(* IEC 61131-3 sources: std_i2980_v2.06_cp053/Source/IMM/ieccontrol/system (part 2) *)

(* ---- ABEnergy.pu ---- *)
(*
@h    ! WARNING !
@h    The Kemro K2 system (including software) only meets category B according to EN 954-1,
@h    thus it is not intended for usage in safety-relevant control applications in the field
@h    of personal safety (e.g. emergency stop).
@h    To implement potentially necessary safety-relevant control tasks, always use additional
@h    external safety devices that are intended for the particular purpose, and meet the necessary
@h    functional safety.
@h    For further information see EN 954-1 (EN ISO 13849-1) and/or the K2-x00 user manual, chapter
@h    "CE conformity, directives and standards".

This AB calculate the energy.

*)

IMPORT_OVER_LISTFILE
 GET_SYNC_REFTO
, GET_TASK_INTERVAL
, GET_MY_FU_NAME
, KSWO_AddVariable
, START_PROCESS_ALGORITHM
, STOP_PROCESS_ALGORITHM
, KSYS_Status_OK
, nHalfAutomatic
, nFullAutomatic
, cCompEnergyMeter
, tnOperationMode
, tyNumberOfDevices
, KSYS_Status
, KSWO_Status

END_IMPORT

ALGORITHM_BLOCK ABEnergy #DUMMY_EDIT_BLOCK

SYSTEM_VAR
 sv_bResetShotCounter : BOOL (* reset shot counter *);
 sv_iProdCounterAct : DINT;
 sv_iShotCounterAct : DINT;
 sv_rEnergyShot : REAL (* energy per shot *);
 sv_rEnergyProduction : REAL (* energy per production *);
 sv_rEnergyPart : REAL (* energy per part *);
 sv_rEnergyShotVolume : REAL (* energy in shot volume *);
 sv_rEnergyPartMass : REAL (* energy in part mass *);
 sv_rPartMass : REAL (* part mass *);
 sv_rHeatingPower : REAL (* heating power *);
 sv_rTotalEnergy : REAL (* total energy *);
 sv_rTotalPower : REAL (* total power *);
 sv_rMotorPower : REAL (* motor power *);
 sv_bResetTotEnergy : BOOL (* reset energy *);
 sv_OperationMode : tnOperationMode;
 sv_bStartSampleMeasure : BOOL;
 sv_rSampleMeasuredEnergy : REAL;
 sv_iAutoStopShotCounter : DINT;
 sv_dMeasuredDuration : TIME (* measured duration in mins  *);
 sv_dSetDuration : TIME (* set duration for sample energy measurement in mins  *);
 sv_rMeasuredPower : REAL (* measured  power *);
 sv_rMeasuredEnergy : REAL (* measured energy *);
 sv_rTotalEnergyCalibrated : REAL (* total energy *);
 sv_rTotalPowerCalibrated : REAL (* total power *);
 sv_rIdlePower : REAL;
 sv_rMeasuredEnergyHMI : REAL;
 sv_NumberOfDevices : tyNumberOfDevices;
 sv_bInitDone : BOOL;
 sv_rEfficiency : REAL;
END_VAR

SYSTEM_OBJECT
 TaskMid : TASK;
 TaskSlow : TASK;
 TaskHeating : TASK;
 TaskInject : TASK;
 PU_Task_7 : TASK;
END_OBJECT

VAR
 mrMotorPower : REAL;
 mprActCushion : REFTO REAL;
 mprCushionZeroPosition : REFTO REAL;
 mrActEnergy : REAL;
 mrTotEnergyLastShot : REAL;
 mrTotEnergyLastPart : REAL;
 mrShotVolume : REAL;
 mrTmpEnergy : REAL;
 mrLastActEnergy : REAL;
 mprHeatingPowerNozzle1 : REFTO REAL;
 mprHeatingPowerMold1 : REFTO REAL;
 mbHeatingPowerNozzle1Linked : BOOL;
 mbHeatingPowerMold1Linked : BOOL;
 mrRecordedEnergy : REAL;
 mbCycleRestarted : BOOL;
 miShotCounter : DINT;
 mrRecordedSampleEnergy : REAL;
 mrActEnergyCalibrated : REAL;
 mrTmpEnergyCalibrated : REAL;
 mbEnergyMeterLinked : BOOL;
 mprMotorPowerSpeedpump : REFTO REAL;
 mprMotorPowerEject : REFTO REAL;
 mprMotorPowerInject : REFTO REAL;
 mprMotorPowerPlast : REFTO REAL;
 mprMotorPowerMold : REFTO REAL;
 mprMotorPowerNozzle : REFTO REAL;
END_VAR

(*
@h    ! WARNING !
@h    The Kemro K2 system (including software) only meets category B according to EN 954-1,
@h    thus it is not intended for usage in safety-relevant control applications in the field
@h    of personal safety (e.g. emergency stop).
@h    To implement potentially necessary safety-relevant control tasks, always use additional
@h    external safety devices that are intended for the particular purpose, and meet the necessary
@h    functional safety.
@h    For further information see EN 954-1 (EN ISO 13849-1) and/or the K2-x00 user manual, chapter
@h    "CE conformity, directives and standards".

This algo initializes for the energy calculation

*)

PROCESS_ALGORITHM paInit ON TaskMid AUTOSTART

VAR
 Status : KSYS_Status;
END_VAR
#BEGIN_EDIT_BLOCK
(**************************************** WARNING ********************************************
 *** The KEBA Kemro K2 System including software is not intended for safety control tasks! ***
 ***                       For further information see Comment tab!                        ***
 *********************************************************************************************)

(*pointer to motor total power speedpump*)
mprMotorPowerSpeedpump := GET_SYNC_REFTO('Pump1.sv_rMotorTotalPower', T#0s, Status);

IF Status <> KSYS_Status_OK  THEN
   mprMotorPowerSpeedpump := GET_SYNC_REFTO('system.sv_rNull', T#0s, Status);
END_IF;

(*pointer to motor power elec.axes*)
mprMotorPowerEject := GET_SYNC_REFTO('Ejector1.sv_rMotorPowerEject', T#0s, Status);
IF Status <> KSYS_Status_OK  THEN
   mprMotorPowerEject := GET_SYNC_REFTO('system.sv_rNull', T#0s, Status);
END_IF;

mprMotorPowerInject:= GET_SYNC_REFTO('Injection1.sv_rMotorPowerInject', T#0s, Status);
IF Status <> KSYS_Status_OK  THEN
   mprMotorPowerInject := GET_SYNC_REFTO('system.sv_rNull', T#0s, Status);
END_IF;

mprMotorPowerPlast:= GET_SYNC_REFTO('Injection1.sv_rMotorPowerPlast', T#0s, Status);
IF Status <> KSYS_Status_OK  THEN
   mprMotorPowerPlast := GET_SYNC_REFTO('system.sv_rNull', T#0s, Status);
END_IF;

mprMotorPowerMold:= GET_SYNC_REFTO('Mold1.sv_rMotorPowerMold', T#0s, Status);
IF Status <> KSYS_Status_OK  THEN
   mprMotorPowerMold := GET_SYNC_REFTO('system.sv_rNull', T#0s, Status);
END_IF;

mprMotorPowerNozzle:= GET_SYNC_REFTO('Nozzle1.sv_rMotorPowerNozzle', T#0s, Status);
IF Status <> KSYS_Status_OK  THEN
   mprMotorPowerNozzle := GET_SYNC_REFTO('system.sv_rNull', T#0s, Status);
END_IF;

mprActCushion := GET_SYNC_REFTO('Injection1.sv_rCushion', T#0s, Status);
mprCushionZeroPosition := GET_SYNC_REFTO('Injection1.sv_rScrewZeroPosition', T#0s, Status);

mprHeatingPowerNozzle1 := GET_SYNC_REFTO('HeatingNozzle1.sv_rActHeatingPower', T#0s, Status);
IF Status = KSYS_Status_OK THEN
   mbHeatingPowerNozzle1Linked := TRUE;
END_IF;
mprHeatingPowerMold1 := GET_SYNC_REFTO('HeatingMold1.sv_rActHeatingPower', T#0s, Status);
IF Status = KSYS_Status_OK THEN
   mbHeatingPowerMold1Linked := TRUE;
END_IF;

STOP_PROCESS_ALGORITHM();

;#END_EDIT_BLOCK END_ALGORITHM

(*
@h    ! WARNING !
@h    The Kemro K2 system (including software) only meets category B according to EN 954-1,
@h    thus it is not intended for usage in safety-relevant control applications in the field
@h    of personal safety (e.g. emergency stop).
@h    To implement potentially necessary safety-relevant control tasks, always use additional
@h    external safety devices that are intended for the particular purpose, and meet the necessary
@h    functional safety.
@h    For further information see EN 954-1 (EN ISO 13849-1) and/or the K2-x00 user manual, chapter
@h    "CE conformity, directives and standards".

This postupdate algorithms calculates the energy per shot and per ccm.

*)

POSTUPDATE_ALGORITHM pCalcEnergyShot ON TaskMid WITH sv_iShotCounterAct

#BEGIN_EDIT_BLOCK
(**************************************** WARNING ********************************************
 *** The KEBA Kemro K2 System including software is not intended for safety control tasks! ***
 ***                       For further information see Comment tab!                        ***
 *********************************************************************************************)

(*Calculation of the energy cosumption per shot*)
sv_rEnergyShot := mrActEnergy - mrTotEnergyLastShot;
mrTotEnergyLastShot := mrActEnergy;

(*Calculation of the energy cosumption per ccm*)
mrShotVolume := mprCushionZeroPosition^ - mprActCushion^;  (*calculate the shot volume*)

IF mrShotVolume <> 0.0 THEN
  sv_rEnergyShotVolume := sv_rEnergyShot / mrShotVolume;
ELSE
  sv_rEnergyShotVolume := 0.0;
END_IF;

//Synchronization to machine cycle
IF mbEnergyMeterLinked THEN
  IF sv_bStartSampleMeasure THEN

  //start the sample measurement
    IF NOT mbCycleRestarted THEN
      mbCycleRestarted := TRUE;
    END_IF;

    //shot counter for the sample measurement
    miShotCounter := miShotCounter + 1;
    END_IF;
END_IF;

;#END_EDIT_BLOCK END_ALGORITHM

(*
@h    ! WARNING !
@h    The Kemro K2 system (including software) only meets category B according to EN 954-1,
@h    thus it is not intended for usage in safety-relevant control applications in the field
@h    of personal safety (e.g. emergency stop).
@h    To implement potentially necessary safety-relevant control tasks, always use additional
@h    external safety devices that are intended for the particular purpose, and meet the necessary
@h    functional safety.
@h    For further information see EN 954-1 (EN ISO 13849-1) and/or the K2-x00 user manual, chapter
@h    "CE conformity, directives and standards".

This AB calculates the energy per production.

*)

POSTUPDATE_ALGORITHM pUpdateEnergyProduction ON TaskMid WITH sv_bResetShotCounter

#BEGIN_EDIT_BLOCK
(**************************************** WARNING ********************************************
 *** The KEBA Kemro K2 System including software is not intended for safety control tasks! ***
 ***                       For further information see Comment tab!                        ***
 *********************************************************************************************)
sv_rEnergyProduction := 0.0;             (*reset the energy per production*)
mrLastActEnergy := mrActEnergy;          (*copy the calculated energy of the last cycle*)

;#END_EDIT_BLOCK END_ALGORITHM

(*
@h    ! WARNING !
@h    The Kemro K2 system (including software) only meets category B according to EN 954-1,
@h    thus it is not intended for usage in safety-relevant control applications in the field
@h    of personal safety (e.g. emergency stop).
@h    To implement potentially necessary safety-relevant control tasks, always use additional
@h    external safety devices that are intended for the particular purpose, and meet the necessary
@h    functional safety.
@h    For further information see EN 954-1 (EN ISO 13849-1) and/or the K2-x00 user manual, chapter
@h    "CE conformity, directives and standards".

This postupdate algorithm calculates the energy per gram.
*)

POSTUPDATE_ALGORITHM pCalcEnergyPart ON TaskMid WITH sv_iProdCounterAct,sv_rPartMass

#BEGIN_EDIT_BLOCK
(**************************************** WARNING ********************************************
 *** The KEBA Kemro K2 System including software is not intended for safety control tasks! ***
 ***                       For further information see Comment tab!                        ***
 *********************************************************************************************)

(*Calculation of the energy cosumption per part*)
sv_rEnergyPart := mrActEnergy - mrTotEnergyLastPart;
mrTotEnergyLastPart := mrActEnergy;

(*Calculation of the energy cosumption in part mass*)
IF sv_rPartMass <> 0.0 THEN
    sv_rEnergyPartMass := sv_rEnergyPart / sv_rPartMass;
ELSE
    sv_rEnergyPartMass := 0.0;
END_IF;

;#END_EDIT_BLOCK END_ALGORITHM

(*
@h    ! WARNING !
@h    The Kemro K2 system (including software) only meets category B according to EN 954-1,
@h    thus it is not intended for usage in safety-relevant control applications in the field
@h    of personal safety (e.g. emergency stop).
@h    To implement potentially necessary safety-relevant control tasks, always use additional
@h    external safety devices that are intended for the particular purpose, and meet the necessary
@h    functional safety.
@h    For further information see EN 954-1 (EN ISO 13849-1) and/or the K2-x00 user manual, chapter
@h    "CE conformity, directives and standards".

This process algorithm calculates the energy.
*)

PROCESS_ALGORITHM paCalcAndMeasure ON TaskHeating

VAR_TEMP
 b : BOOL;
END_VAR

VAR
 rHeatingPower : REAL;
 dCycleTime : TIME;
 bInitDone : BOOL;
 rCycleTime : REAL;
END_VAR
#BEGIN_EDIT_BLOCK
(**************************************** WARNING ********************************************
 *** The KEBA Kemro K2 System including software is not intended for safety control tasks! ***
 ***                       For further information see Comment tab!                        ***
 *********************************************************************************************)

(* Cycle time *)
IF NOT bInitDone THEN
   dCycleTime := GET_TASK_INTERVAL();
   rCycleTime := (LINT_TO_REAL(TIME_TO_LINT(dCycleTime))) / 1000000.0;
   bInitDone := TRUE;
END_IF;

(* Motor power estimated [kW] *)
mrMotorPower :=  mprMotorPowerSpeedpump^ +  mprMotorPowerEject^ +  mprMotorPowerInject^ +  mprMotorPowerPlast^ + mprMotorPowerMold^ + mprMotorPowerNozzle^;
b := WRITE_SVREAL_DIRECT(sv_rMotorPower, mrMotorPower);

(* Heat power estimated [W] *)
rHeatingPower := 0.0;
IF mbHeatingPowerNozzle1Linked THEN
   rHeatingPower := rHeatingPower + mprHeatingPowerNozzle1^;
END_IF;
IF mbHeatingPowerMold1Linked THEN
   rHeatingPower := rHeatingPower + mprHeatingPowerMold1^;
END_IF;
b := WRITE_SVREAL_DIRECT(sv_rHeatingPower, rHeatingPower);

(* Total power [kW] *)
IF mbEnergyMeterLinked THEN
   //Calculate the total power from measured total power
   b := WRITE_SVREAL_DIRECT(sv_rTotalPower, (sv_rMeasuredPower / 1000.0));
ELSE
   b := WRITE_SVREAL_DIRECT(sv_rTotalPower, (((rHeatingPower + sv_rIdlePower) / 1000.0 + mrMotorPower) / sv_rEfficiency));
END_IF;

(* Energy *)
IF mbEnergyMeterLinked THEN
   (* Total energy from power meter [kwh] *)
   sv_rTotalEnergy := (sv_rMeasuredEnergy - mrRecordedEnergy) / 1000.0; //measured value in Wh
   mrActEnergy := sv_rTotalEnergy;
   b := WRITE_SVREAL_DIRECT(sv_rMeasuredEnergyHMI, (sv_rMeasuredEnergy / 1000.0));

   (* Calculate the energy per production [kwh] *)
   IF sv_OperationMode >= nHalfAutomatic THEN
      b := WRITE_SVREAL_DIRECT(sv_rEnergyProduction, ((mrActEnergy - mrLastActEnergy) / 1000.0));
   END_IF;
ELSE
   (* Integration of power = Energy [kWs] *)
   mrActEnergy := mrTmpEnergy + sv_rTotalPower * rCycleTime;
   mrTmpEnergy := mrActEnergy;

   (* Calculate the energy per production [kwh] *)
   IF sv_OperationMode >= nHalfAutomatic THEN
      b := WRITE_SVREAL_DIRECT(sv_rEnergyProduction, ((mrActEnergy - mrLastActEnergy) / 3600.0));
   END_IF;

   (* Consumption of energy [kwh] *)
   sv_rTotalEnergy := (mrActEnergy / 3600.0 + mrRecordedEnergy);
END_IF;

(* Calibration *)
IF mbEnergyMeterLinked THEN
   (* Power calibration *)
   b := WRITE_SVREAL_DIRECT(sv_rTotalPowerCalibrated, ((sv_rMotorPower + (sv_rHeatingPower + sv_rIdlePower) / 1000.0) / sv_rEfficiency));

   (* Energy calibration *)
   mrActEnergyCalibrated := mrTmpEnergyCalibrated + sv_rTotalPowerCalibrated * rCycleTime;
   mrTmpEnergyCalibrated := mrActEnergyCalibrated;
   b := WRITE_SVREAL_DIRECT(sv_rTotalEnergyCalibrated, (mrActEnergyCalibrated / 3600.0));
END_IF;

;#END_EDIT_BLOCK END_ALGORITHM

(*
@h    ! WARNING !
@h    The Kemro K2 system (including software) only meets category B according to EN 954-1,
@h    thus it is not intended for usage in safety-relevant control applications in the field
@h    of personal safety (e.g. emergency stop).
@h    To implement potentially necessary safety-relevant control tasks, always use additional
@h    external safety devices that are intended for the particular purpose, and meet the necessary
@h    functional safety.
@h    For further information see EN 954-1 (EN ISO 13849-1) and/or the K2-x00 user manual, chapter
@h    "CE conformity, directives and standards".

This postupdate algorithm resets the energy calculation.
*)

POSTUPDATE_ALGORITHM pResetTotalEnergy ON TaskMid WITH sv_bResetTotEnergy

#BEGIN_EDIT_BLOCK
(**************************************** WARNING ********************************************
 *** The KEBA Kemro K2 System including software is not intended for safety control tasks! ***
 ***                       For further information see Comment tab!                        ***
 *********************************************************************************************)
(*reset the energy calculator*)
IF sv_bResetTotEnergy THEN
   //when power meter is used, record the last measured total energy,
   //and calculate always the difference between the actual measured value and recorded value
   //when estimation is used, integration of power with initial value 0 would be restarted
   IF mbEnergyMeterLinked THEN
     mrRecordedEnergy := sv_rMeasuredEnergy;
   ELSE
     mrRecordedEnergy := 0.0;
   END_IF;

   mrActEnergy := 0.0;
   mrTmpEnergy := 0.0;
   sv_rTotalEnergy := 0.0;
   mrLastActEnergy := 0.0;
   mrTotEnergyLastShot := 0.0;
   mrTotEnergyLastPart := 0.0;
   sv_bResetTotEnergy := FALSE;

   //calibration
   IF mbEnergyMeterLinked THEN
     mrActEnergyCalibrated := 0.0;
     mrTmpEnergyCalibrated := 0.0;
     sv_rTotalEnergyCalibrated := 0.0;
   END_IF;
END_IF;

;#END_EDIT_BLOCK END_ALGORITHM

PROCESS_ALGORITHM paInitDebugMeasurement ON TaskSlow AUTOSTART

VAR
 fuName : STRING(255);
 variableName : STRING(255);
 swoState : KSWO_Status;
END_VAR
#BEGIN_EDIT_BLOCK
(**************************************** WARNING ********************************************
 *** The KEBA Kemro K2 System including software is not intended for safety control tasks! ***
 ***                       For further information see Comment tab!                        ***
 *********************************************************************************************)
fuName := GET_MY_FU_NAME();
variableName := CONCAT(fuName,'.rMotorPowerCalc kW');
swoState := KSWO_AddVariable( Task := TaskInject,
                              Name := variableName,
                              Variable := sv_rMotorPower);
variableName := CONCAT(fuName,'.rTotalEnergyMeasured kWh');
swoState := KSWO_AddVariable( Task := TaskInject,
                              Name := variableName,
                              Variable := sv_rTotalEnergy);
variableName := CONCAT(fuName,'.rTotalEnergyCalibrated kWh');
swoState := KSWO_AddVariable( Task := TaskInject,
                              Name := variableName,
                              Variable := sv_rTotalEnergyCalibrated);
variableName := CONCAT(fuName,'.rTotalPower kW');
swoState := KSWO_AddVariable( Task := TaskInject,
                              Name := variableName,
                              Variable := sv_rTotalPower);
STOP_PROCESS_ALGORITHM();

;#END_EDIT_BLOCK END_ALGORITHM

(*
@h    ! WARNING !
@h    The Kemro K2 system (including software) only meets category B according to EN 954-1,
@h    thus it is not intended for usage in safety-relevant control applications in the field
@h    of personal safety (e.g. emergency stop).
@h    To implement potentially necessary safety-relevant control tasks, always use additional
@h    external safety devices that are intended for the particular purpose, and meet the necessary
@h    functional safety.
@h    For further information see EN 954-1 (EN ISO 13849-1) and/or the K2-x00 user manual, chapter
@h    "CE conformity, directives and standards".

This postppdate algorithm resets the temp variables for sum.

*)

POSTUPDATE_ALGORITHM pInitRecord ON TaskInject WITH sv_OperationMode

#BEGIN_EDIT_BLOCK
(**************************************** WARNING ********************************************
 *** The KEBA Kemro K2 System including software is not intended for safety control tasks! ***
 ***                       For further information see Comment tab!                        ***
 *********************************************************************************************)
(*Reset the last sum*)
IF sv_OperationMode = nFullAutomatic THEN
    mrTotEnergyLastShot := 0.0;
    mrTotEnergyLastPart := 0.0;
END_IF;

;#END_EDIT_BLOCK END_ALGORITHM

POSTUPDATE_ALGORITHM pSampleMeasure ON PU_Task_7 WITH sv_bStartSampleMeasure

#BEGIN_EDIT_BLOCK
//start the sample measurement
IF sv_bStartSampleMeasure THEN
  START_PROCESS_ALGORITHM(paSampleMeasure);
END_IF;

;#END_EDIT_BLOCK END_ALGORITHM

PROCESS_ALGORITHM paSampleMeasure ON TaskHeating

VAR
 bLastMeasurementInitialized : BOOL;
 rMeasuredDuration : REAL;
 dCycleTime : TIME;
 rCycleTime : REAL;
 rSetDuration : REAL;
END_VAR
#BEGIN_EDIT_BLOCK
IF mbCycleRestarted THEN

  //Initialization of measurement
  IF NOT bLastMeasurementInitialized THEN
    bLastMeasurementInitialized := TRUE;
    mrRecordedSampleEnergy := sv_rMeasuredEnergy;  //read the latest measured energy
    miShotCounter := 0;                         //reset the shotcounter for sampling
    rMeasuredDuration := 0.0;                   //reset the duration for sampling
    dCycleTime := GET_TASK_INTERVAL();
    rCycleTime := (LINT_TO_REAL(TIME_TO_LINT(dCycleTime))) / 1.0e6;  //in seconds
    rSetDuration := LINT_TO_REAL(TIME_TO_LINT(sv_dSetDuration)) / 1.0e6;   //set duration in seconds
  END_IF;

  //Energy consumption from starting the sampling
  sv_rSampleMeasuredEnergy := (sv_rMeasuredEnergy - mrRecordedSampleEnergy) / 1.0e3;

  rMeasuredDuration := rMeasuredDuration + rCycleTime;
  sv_dMeasuredDuration := LINT_TO_TIME(REAL_TO_LINT(rMeasuredDuration * 1.0e6));    //in mins

  //Auto-Stop dependant on shot counter and set measurement duration
  //Automatically stopped when shot counter or duration first is reached
  IF ((miShotCounter >= sv_iAutoStopShotCounter) AND (sv_iAutoStopShotCounter <> 0))
                             OR ((rMeasuredDuration >= rSetDuration) AND (rSetDuration <> 0.0)) OR (NOT sv_bStartSampleMeasure) THEN

      mbCycleRestarted := FALSE;
    sv_bStartSampleMeasure := FALSE;
    bLastMeasurementInitialized := FALSE;

    STOP_PROCESS_ALGORITHM();
  END_IF;
ELSE  //waiting for the start of next cycle
  sv_rSampleMeasuredEnergy := 0.0; //reset the measurement
  sv_dMeasuredDuration := t#0s;    //reset the timer
END_IF;

;#END_EDIT_BLOCK END_ALGORITHM

POSTUPDATE_ALGORITHM pInit ON PU_Task_7 WITH sv_bInitDone

#BEGIN_EDIT_BLOCK
//Energy meter is linked
IF sv_NumberOfDevices[cCompEnergyMeter] <> 0 THEN
  mbEnergyMeterLinked := TRUE;
END_IF;

// Calculate/Measure power/energy cyclically
START_PROCESS_ALGORITHM(paCalcAndMeasure);

IF NOT mbEnergyMeterLinked THEN
  mrRecordedEnergy := sv_rTotalEnergy;
ELSE
  mrRecordedEnergy := sv_rMeasuredEnergy; //initialization
END_IF;

;#END_EDIT_BLOCK END_ALGORITHM

END_ALGORITHM_BLOCK

#END_OF_IEC_PART

@Puma @IecEditor 6 128 @Pou 25
@@@BEG_Comment@@@
@h    ! WARNING !
@h    The Kemro K2 system (including software) only meets category B according to EN 954-1,
@h    thus it is not intended for usage in safety-relevant control applications in the field
@h    of personal safety (e.g. emergency stop).
@h    To implement potentially necessary safety-relevant control tasks, always use additional
@h    external safety devices that are intended for the particular purpose, and meet the necessary
@h    functional safety.
@h    For further information see EN 954-1 (EN ISO 13849-1) and/or the K2-x00 user manual, chapter
@h    "CE conformity, directives and standards".

This AB calculate the energy.

@@@END_Comment@@@

@BEG_Contents

@BEG_Func
@RT(17)FuncTreeContainer
6
@Var @RT(14)GET_SYNC_REFTO @RT(0) @T @T @DERIVED 0 @F @RT(22)KEBA_STANDARD_FUNCTION @F
@T
@BEG_Attrib
0 @RT(0) @RT(0)
@END_Attrib
1 1 @F @F @F @F

@Var @RT(17)GET_TASK_INTERVAL @RT(0) @T @T @DERIVED 0 @F @RT(22)KEBA_STANDARD_FUNCTION @F
@T
@BEG_Attrib
0 @RT(0) @RT(0)
@END_Attrib
1 1 @F @F @F @F

@Var @RT(14)GET_MY_FU_NAME @RT(0) @T @T @DERIVED 0 @F @RT(22)KEBA_STANDARD_FUNCTION @F
@T
@BEG_Attrib
0 @RT(0) @RT(0)
@END_Attrib
1 1 @F @F @F @F

@Var @RT(16)KSWO_AddVariable @RT(0) @T @T @DERIVED 0 @F @RT(22)KEBA_STANDARD_FUNCTION @F
@T
@BEG_Attrib
0 @RT(0) @RT(0)
@END_Attrib
1 1 @F @F @F @F

@Var @RT(23)START_PROCESS_ALGORITHM @RT(0) @T @T @DERIVED 0 @F @RT(23)KEBA_STANDARD_PROCEDURE @F
@T
@BEG_Attrib
0 @RT(0) @RT(0)
@END_Attrib
1 1 @F @F @F @F

@Var @RT(22)STOP_PROCESS_ALGORITHM @RT(0) @T @T @DERIVED 0 @F @RT(23)KEBA_STANDARD_PROCEDURE @F
@T
@BEG_Attrib
0 @RT(0) @RT(0)
@END_Attrib
1 1 @F @F @F @F

@END_Func

@BEG_Const
@RT(18)ConstTreeContainer
4
@Var @RT(14)KSYS_Status_OK @RT(0) @T @T @DERIVED 0 @F @RT(11)KSYS_Status @F
@T
@BEG_Attrib
0 @RT(1)1 @RT(0)
@END_Attrib
1 1 @F @F @F @F

@Var @RT(14)nHalfAutomatic @RT(0) @T @T @DERIVED 0 @F @RT(15)tnOperationMode @F
@T
@BEG_Attrib
0 @RT(1)2 @RT(34)confirmation every cycle necessary
@END_Attrib
1 1 @F @F @F @F

@Var @RT(14)nFullAutomatic @RT(0) @T @T @DERIVED 0 @F @RT(15)tnOperationMode @F
@T
@BEG_Attrib
0 @RT(1)3 @RT(47)confirmation only for the first cycle necessary
@END_Attrib
1 1 @F @F @F @F

@Var @RT(16)cCompEnergyMeter @RT(0) @T @F @DT @RT(4)DINT @RT(0) @T @T @BASIC 0 @F
@F @F
@T
@BEG_Attrib
0 @RT(3)157 @RT(22)Component Energy meter
@END_Attrib
1 1 @F @F @F @F

@END_Const

@BEG_Export

@BEG_Kind
@ALGORITHM_BLOCK @RT(8)ABEnergy @STRUCTURED_TEXT
@RT(0) @RT(0) @RT(0)
@END_Kind

@BEG_Dcl
@RT(16)DclTreeContainer
60
@Var @RT(20)sv_bResetShotCounter @RT(0) @T @F @DT @RT(4)BOOL @RT(0) @T @T @BASIC 0 @F
@F @F
@T
@BEG_Attrib
3 @RT(0) @RT(18)reset shot counter @RT(0)
@END_Attrib
1 8 @F @F @F @F

@Var @RT(18)sv_iProdCounterAct @RT(0) @T @F @DT @RT(4)DINT @RT(0) @T @T @BASIC 0 @F
@F @F
@T
@BEG_Attrib
3 @RT(0) @RT(0) @RT(0)
@END_Attrib
1 8 @F @F @F @F

@Var @RT(18)sv_iShotCounterAct @RT(0) @T @F @DT @RT(4)DINT @RT(0) @T @T @BASIC 0 @F
@F @F
@T
@BEG_Attrib
3 @RT(0) @RT(0) @RT(0)
@END_Attrib
1 8 @F @F @F @F

@Var @RT(14)sv_rEnergyShot @RT(0) @T @F @DT @RT(4)REAL @RT(0) @T @T @BASIC 0 @F
@F @F
@T
@BEG_Attrib
3 @RT(0) @RT(15)energy per shot @RT(0)
@END_Attrib
1 8 @F @F @F @F

@Var @RT(20)sv_rEnergyProduction @RT(0) @T @F @DT @RT(4)REAL @RT(0) @T @T @BASIC 0 @F
@F @F
@T
@BEG_Attrib
3 @RT(0) @RT(21)energy per production @RT(0)
@END_Attrib
1 8 @F @F @F @F

@Var @RT(14)sv_rEnergyPart @RT(0) @T @F @DT @RT(4)REAL @RT(0) @T @T @BASIC 0 @F
@F @F
@T
@BEG_Attrib
3 @RT(0) @RT(15)energy per part @RT(0)
@END_Attrib
1 8 @F @F @F @F

@Var @RT(20)sv_rEnergyShotVolume @RT(0) @T @F @DT @RT(4)REAL @RT(0) @T @T @BASIC 0 @F
@F @F
@T
@BEG_Attrib
3 @RT(0) @RT(21)energy in shot volume @RT(0)
@END_Attrib
1 8 @F @F @F @F

@Var @RT(18)sv_rEnergyPartMass @RT(0) @T @F @DT @RT(4)REAL @RT(0) @T @T @BASIC 0 @F
@F @F
@T
@BEG_Attrib
3 @RT(0) @RT(19)energy in part mass @RT(0)
@END_Attrib
1 8 @F @F @F @F

@Var @RT(12)sv_rPartMass @RT(0) @T @F @DT @RT(4)REAL @RT(0) @T @T @BASIC 0 @F
@F @F
@T
@BEG_Attrib
3 @RT(0) @RT(9)part mass @RT(0)
@END_Attrib
1 8 @F @F @F @F

@Var @RT(16)sv_rHeatingPower @RT(0) @T @F @DT @RT(4)REAL @RT(0) @T @T @BASIC 0 @F
@F @F
@T
@BEG_Attrib
3 @RT(0) @RT(13)heating power @RT(0)
@END_Attrib
1 8 @F @F @F @F

@Var @RT(15)sv_rTotalEnergy @RT(0) @T @F @DT @RT(4)REAL @RT(0) @T @T @BASIC 0 @F
@F @F
@T
@BEG_Attrib
3 @RT(0) @RT(12)total energy @RT(0)
@END_Attrib
1 8 @F @F @F @F

@Var @RT(14)sv_rTotalPower @RT(0) @T @F @DT @RT(4)REAL @RT(0) @T @T @BASIC 0 @F
@F @F
@T
@BEG_Attrib
3 @RT(0) @RT(11)total power @RT(0)
@END_Attrib
1 8 @F @F @F @F

@Var @RT(14)sv_rMotorPower @RT(0) @T @F @DT @RT(4)REAL @RT(0) @T @T @BASIC 0 @F
@F @F
@T
@BEG_Attrib
3 @RT(0) @RT(11)motor power @RT(0)
@END_Attrib
1 8 @F @F @F @F

@Var @RT(18)sv_bResetTotEnergy @RT(0) @T @F @DT @RT(4)BOOL @RT(0) @T @T @BASIC 0 @F
@F @F
@T
@BEG_Attrib
3 @RT(0) @RT(12)reset energy @RT(0)
@END_Attrib
1 8 @F @F @F @F

@Var @RT(16)sv_OperationMode @RT(0) @T @T @DERIVED 0 @T @T @DT @RT(15)tnOperationMode @RT(0) @T @T @UNKNOWN 0 @F
@F @F
@T
@BEG_Attrib
3 @RT(0) @RT(0) @RT(0)
@END_Attrib
1 8 @F @F @F @F

@Var @RT(7)TaskMid @RT(0) @T @F @DT @RT(4)TASK @RT(0) @T @T @BASIC 0 @F
@F @F
@T
@BEG_Attrib
3 @RT(0) @RT(0) @RT(0)
@END_Attrib
1 7 @F @F @F @F

@Var @RT(8)TaskSlow @RT(0) @T @F @DT @RT(4)TASK @RT(0) @T @T @BASIC 0 @F
@F @F
@T
@BEG_Attrib
3 @RT(0) @RT(0) @RT(0)
@END_Attrib
1 7 @F @F @F @F

@Var @RT(11)TaskHeating @RT(0) @T @T @RENAMED 0 @T @T @DT @RT(4)TASK @RT(0) @T @T @BASIC 0 @F
@F @F
@T
@BEG_Attrib
3 @RT(0) @RT(0) @RT(0)
@END_Attrib
1 7 @F @F @F @F

@Var @RT(10)TaskInject @RT(0) @T @F @DT @RT(4)TASK @RT(0) @T @T @BASIC 0 @F
@F @F
@T
@BEG_Attrib
3 @RT(0) @RT(0) @RT(0)
@END_Attrib
1 7 @F @F @F @F

@Var @RT(12)mrMotorPower @RT(0) @T @F @DT @RT(4)REAL @RT(0) @T @T @BASIC 0 @F
@F @F
@T
@BEG_Attrib
3 @RT(0) @RT(0) @RT(0)
@END_Attrib
1 0 @F @F @F @F

@Var @RT(13)mprActCushion @RT(0) @T @T @REFTO 0 @T @DT @RT(4)REAL @RT(0) @T @T @BASIC 0 @F
@F @F
@T
@BEG_Attrib
3 @RT(0) @RT(0) @RT(0)
@END_Attrib
1 0 @F @F @F @F

@Var @RT(22)mprCushionZeroPosition @RT(0) @T @T @REFTO 0 @T @DT @RT(4)REAL @RT(0) @T @T @BASIC 0 @F
@F @F
@T
@BEG_Attrib
3 @RT(0) @RT(0) @RT(0)
@END_Attrib
1 0 @F @F @F @F

@Var @RT(11)mrActEnergy @RT(0) @T @F @DT @RT(4)REAL @RT(0) @T @T @BASIC 0 @F
@F @F
@T
@BEG_Attrib
3 @RT(0) @RT(0) @RT(0)
@END_Attrib
1 0 @F @F @F @F

@Var @RT(19)mrTotEnergyLastShot @RT(0) @T @F @DT @RT(4)REAL @RT(0) @T @T @BASIC 0 @F
@F @F
@T
@BEG_Attrib
3 @RT(0) @RT(0) @RT(0)
@END_Attrib
1 0 @F @F @F @F

@Var @RT(19)mrTotEnergyLastPart @RT(0) @T @F @DT @RT(4)REAL @RT(0) @T @T @BASIC 0 @F
@F @F
@T
@BEG_Attrib
3 @RT(0) @RT(0) @RT(0)
@END_Attrib
1 0 @F @F @F @F

@Var @RT(12)mrShotVolume @RT(0) @T @F @DT @RT(4)REAL @RT(0) @T @T @BASIC 0 @F
@F @F
@T
@BEG_Attrib
3 @RT(0) @RT(0) @RT(0)
@END_Attrib
1 0 @F @F @F @F

@Var @RT(11)mrTmpEnergy @RT(0) @T @F @DT @RT(4)REAL @RT(0) @T @T @BASIC 0 @F
@F @F
@T
@BEG_Attrib
3 @RT(0) @RT(0) @RT(0)
@END_Attrib
1 0 @F @F @F @F

@Var @RT(15)mrLastActEnergy @RT(0) @T @F @DT @RT(4)REAL @RT(0) @T @T @BASIC 0 @F
@F @F
@T
@BEG_Attrib
3 @RT(0) @RT(0) @RT(0)
@END_Attrib
1 0 @F @F @F @F

@Var @RT(22)mprHeatingPowerNozzle1 @RT(0) @T @T @REFTO 0 @T @DT @RT(4)REAL @RT(0) @T @T @BASIC 0 @F
@F @F
@T
@BEG_Attrib
3 @RT(0) @RT(0) @RT(0)
@END_Attrib
1 0 @F @F @F @F

@Var @RT(20)mprHeatingPowerMold1 @RT(0) @T @T @REFTO 0 @T @DT @RT(4)REAL @RT(0) @T @T @BASIC 0 @F
@F @F
@T
@BEG_Attrib
3 @RT(0) @RT(0) @RT(0)
@END_Attrib
1 0 @F @F @F @F

@Var @RT(27)mbHeatingPowerNozzle1Linked @RT(0) @T @F @DT @RT(4)BOOL @RT(0) @T @T @BASIC 0 @F
@F @F
@T
@BEG_Attrib
3 @RT(0) @RT(0) @RT(0)
@END_Attrib
1 0 @F @F @F @F

@Var @RT(25)mbHeatingPowerMold1Linked @RT(0) @T @F @DT @RT(4)BOOL @RT(0) @T @T @BASIC 0 @F
@F @F
@T
@BEG_Attrib
3 @RT(0) @RT(0) @RT(0)
@END_Attrib
1 0 @F @F @F @F

@Var @RT(16)mrRecordedEnergy @RT(0) @T @F @DT @RT(4)REAL @RT(0) @T @T @BASIC 0 @F
@F @F
@T
@BEG_Attrib
3 @RT(0) @RT(0) @RT(0)
@END_Attrib
1 0 @F @F @F @F

@Var @RT(9)PU_Task_7 @RT(0) @T @T @RENAMED 0 @T @T @DT @RT(4)TASK @RT(0) @T @T @BASIC 0 @F
@F @F
@T
@BEG_Attrib
3 @RT(0) @RT(0) @RT(0)
@END_Attrib
1 7 @F @F @F @F

@Var @RT(22)sv_bStartSampleMeasure @RT(0) @T @T @RENAMED 0 @T @T @DT @RT(4)BOOL @RT(0) @T @T @BASIC 0 @F
@F @F
@T
@BEG_Attrib
3 @RT(0) @RT(0) @RT(0)
@END_Attrib
1 8 @F @F @F @F

@Var @RT(16)mbCycleRestarted @RT(0) @T @T @RENAMED 0 @T @T @DT @RT(4)BOOL @RT(0) @T @T @BASIC 0 @F
@F @F
@T
@BEG_Attrib
3 @RT(0) @RT(0) @RT(0)
@END_Attrib
1 0 @F @F @F @F

@Var @RT(24)sv_rSampleMeasuredEnergy @RT(0) @T @T @RENAMED 0 @T @T @DT @RT(4)REAL @RT(0) @T @T @BASIC 0 @F
@F @F
@T
@BEG_Attrib
3 @RT(0) @RT(0) @RT(0)
@END_Attrib
1 8 @F @F @F @F

@Var @RT(23)sv_iAutoStopShotCounter @RT(0) @T @T @RENAMED 0 @T @T @DT @RT(4)DINT @RT(0) @T @T @BASIC 0 @F
@F @F
@T
@BEG_Attrib
3 @RT(0) @RT(0) @RT(0)
@END_Attrib
1 8 @F @F @F @F

@Var @RT(20)sv_dMeasuredDuration @RT(0) @T @F @DT @RT(4)TIME @RT(0) @T @T @BASIC 0 @F
@F @F
@T
@BEG_Attrib
3 @RT(0) @RT(26)measured duration in mins  @RT(0)
@END_Attrib
1 8 @F @F @F @F

@Var @RT(15)sv_dSetDuration @RT(0) @T @F @DT @RT(4)TIME @RT(0) @T @T @BASIC 0 @F
@F @F
@T
@BEG_Attrib
3 @RT(0) @RT(51)set duration for sample energy measurement in mins  @RT(0)
@END_Attrib
1 8 @F @F @F @F

@Var @RT(17)sv_rMeasuredPower @RT(0) @T @F @DT @RT(4)REAL @RT(0) @T @T @BASIC 0 @F
@F @F
@T
@BEG_Attrib
3 @RT(0) @RT(15)measured  power @RT(0)
@END_Attrib
1 8 @F @F @F @F

@Var @RT(18)sv_rMeasuredEnergy @RT(0) @T @F @DT @RT(4)REAL @RT(0) @T @T @BASIC 0 @F
@F @F
@T
@BEG_Attrib
3 @RT(0) @RT(15)measured energy @RT(0)
@END_Attrib
1 8 @F @F @F @F

@Var @RT(13)miShotCounter @RT(0) @T @F @DT @RT(4)DINT @RT(0) @T @T @BASIC 0 @F
@F @F
@T
@BEG_Attrib
3 @RT(0) @RT(0) @RT(0)
@END_Attrib
1 0 @F @F @F @F

@Var @RT(22)mrRecordedSampleEnergy @RT(0) @T @T @RENAMED 0 @T @T @DT @RT(4)REAL @RT(0) @T @T @BASIC 0 @F
@F @F
@T
@BEG_Attrib
3 @RT(0) @RT(0) @RT(0)
@END_Attrib
1 0 @F @F @F @F

@Var @RT(21)mrActEnergyCalibrated @RT(0) @T @T @RENAMED 0 @T @T @DT @RT(4)REAL @RT(0) @T @T @BASIC 0 @F
@F @F
@T
@BEG_Attrib
3 @RT(0) @RT(0) @RT(0)
@END_Attrib
1 0 @F @F @F @F

@Var @RT(21)mrTmpEnergyCalibrated @RT(0) @T @T @RENAMED 0 @T @T @DT @RT(4)REAL @RT(0) @T @T @BASIC 0 @F
@F @F
@T
@BEG_Attrib
3 @RT(0) @RT(0) @RT(0)
@END_Attrib
1 0 @F @F @F @F

@Var @RT(25)sv_rTotalEnergyCalibrated @RT(0) @T @F @DT @RT(4)REAL @RT(0) @T @T @BASIC 0 @F
@F @F
@T
@BEG_Attrib
3 @RT(0) @RT(12)total energy @RT(0)
@END_Attrib
1 8 @F @F @F @F

@Var @RT(24)sv_rTotalPowerCalibrated @RT(0) @T @F @DT @RT(4)REAL @RT(0) @T @T @BASIC 0 @F
@F @F
@T
@BEG_Attrib
3 @RT(0) @RT(11)total power @RT(0)
@END_Attrib
1 8 @F @F @F @F

@Var @RT(13)sv_rIdlePower @RT(0) @T @F @DT @RT(4)REAL @RT(0) @T @T @BASIC 0 @F
@F @F
@T
@BEG_Attrib
3 @RT(0) @RT(0) @RT(0)
@END_Attrib
1 8 @F @F @F @F

@Var @RT(21)sv_rMeasuredEnergyHMI @RT(0) @T @T @RENAMED 0 @T @T @DT @RT(4)REAL @RT(0) @T @T @BASIC 0 @F
@F @F
@T
@BEG_Attrib
3 @RT(0) @RT(0) @RT(0)
@END_Attrib
1 8 @F @F @F @F

@Var @RT(18)sv_NumberOfDevices @RT(0) @T @T @DERIVED 0 @T @T @DT @RT(17)tyNumberOfDevices @RT(0) @T @T @UNKNOWN 0 @F
@F @F
@T
@BEG_Attrib
3 @RT(0) @RT(0) @RT(0)
@END_Attrib
1 8 @F @F @F @F

@Var @RT(12)sv_bInitDone @RT(0) @T @T @RENAMED 0 @T @T @DT @RT(4)BOOL @RT(0) @T @T @BASIC 0 @F
@F @F
@T
@BEG_Attrib
3 @RT(0) @RT(0) @RT(0)
@END_Attrib
1 8 @F @F @F @F

@Var @RT(14)sv_rEfficiency @RT(0) @T @F @DT @RT(4)REAL @RT(0) @T @T @BASIC 0 @F
@F @F
@T
@BEG_Attrib
3 @RT(0) @RT(0) @RT(0)
@END_Attrib
1 8 @F @F @F @F

@Var @RT(19)mbEnergyMeterLinked @RT(0) @T @F @DT @RT(4)BOOL @RT(0) @T @T @BASIC 0 @F
@F @F
@T
@BEG_Attrib
3 @RT(0) @RT(0) @RT(0)
@END_Attrib
1 0 @F @F @F @F

@Var @RT(22)mprMotorPowerSpeedpump @RT(0) @T @T @REFTO 0 @T @DT @RT(4)REAL @RT(0) @T @T @BASIC 0 @F
@F @F
@T
@BEG_Attrib
3 @RT(0) @RT(0) @RT(0)
@END_Attrib
1 0 @F @F @F @F

@Var @RT(18)mprMotorPowerEject @RT(0) @T @T @REFTO 0 @T @DT @RT(4)REAL @RT(0) @T @T @BASIC 0 @F
@F @F
@T
@BEG_Attrib
3 @RT(0) @RT(0) @RT(0)
@END_Attrib
1 0 @F @F @F @F

@Var @RT(19)mprMotorPowerInject @RT(0) @T @T @REFTO 0 @T @DT @RT(4)REAL @RT(0) @T @T @BASIC 0 @F
@F @F
@T
@BEG_Attrib
3 @RT(0) @RT(0) @RT(0)
@END_Attrib
1 0 @F @F @F @F

@Var @RT(18)mprMotorPowerPlast @RT(0) @T @T @REFTO 0 @T @DT @RT(4)REAL @RT(0) @T @T @BASIC 0 @F
@F @F
@T
@BEG_Attrib
3 @RT(0) @RT(0) @RT(0)
@END_Attrib
1 0 @F @F @F @F

@Var @RT(17)mprMotorPowerMold @RT(0) @T @T @REFTO 0 @T @DT @RT(4)REAL @RT(0) @T @T @BASIC 0 @F
@F @F
@T
@BEG_Attrib
3 @RT(0) @RT(0) @RT(0)
@END_Attrib
1 0 @F @F @F @F

@Var @RT(19)mprMotorPowerNozzle @RT(0) @T @T @REFTO 0 @T @DT @RT(4)REAL @RT(0) @T @T @BASIC 0 @F
@F @F
@T
@BEG_Attrib
3 @RT(0) @RT(0) @RT(0)
@END_Attrib
1 0 @F @F @F @F

@END_Dcl

@END_Export

@BEG_Body

11

@BEG_Export

@BEG_Algo
@PROCESS_ALGORITHM @RT(6)paInit @STRUCTURED_TEXT
@RT(0) @RT(0) @RT(7)TaskMid @T @F
@END_Algo

@BEG_Dcl
@RT(16)DclTreeContainer
1
@Var @RT(6)Status @RT(0) @T @T @DERIVED 0 @T @T @DT @RT(11)KSYS_Status @RT(0) @T @T @UNKNOWN 0 @F
@F @F
@T
@BEG_Attrib
3 @RT(0) @RT(0) @RT(0)
@END_Attrib
1 0 @F @F @F @F

@END_Dcl

@END_Export

@BEG_Export

@BEG_Algo
@POSTUPDATE_ALGORITHM @RT(15)pCalcEnergyShot @STRUCTURED_TEXT
@RT(0) @RT(18)sv_iShotCounterAct @RT(7)TaskMid @F @F
@END_Algo

@BEG_Dcl
@RT(16)DclTreeContainer
0
@END_Dcl

@END_Export

@BEG_Export

@BEG_Algo
@POSTUPDATE_ALGORITHM @RT(23)pUpdateEnergyProduction @STRUCTURED_TEXT
@RT(0) @RT(20)sv_bResetShotCounter @RT(7)TaskMid @F @F
@END_Algo

@BEG_Dcl
@RT(16)DclTreeContainer
0
@END_Dcl

@END_Export

@BEG_Export

@BEG_Algo
@POSTUPDATE_ALGORITHM @RT(15)pCalcEnergyPart @STRUCTURED_TEXT
@RT(0) @RT(31)sv_iProdCounterAct,sv_rPartMass @RT(7)TaskMid @F @F
@END_Algo

@BEG_Dcl
@RT(16)DclTreeContainer
0
@END_Dcl

@END_Export

@BEG_Export

@BEG_Algo
@PROCESS_ALGORITHM @RT(16)paCalcAndMeasure @STRUCTURED_TEXT
@RT(0) @RT(0) @RT(11)TaskHeating @F @F
@END_Algo

@BEG_Dcl
@RT(16)DclTreeContainer
5
@Var @RT(13)rHeatingPower @RT(0) @T @F @DT @RT(4)REAL @RT(0) @T @T @BASIC 0 @F
@F @F
@T
@BEG_Attrib
3 @RT(0) @RT(0) @RT(0)
@END_Attrib
1 0 @F @F @F @F

@Var @RT(10)dCycleTime @RT(0) @T @F @DT @RT(4)TIME @RT(0) @T @T @BASIC 0 @F
@F @F
@T
@BEG_Attrib
3 @RT(0) @RT(0) @RT(0)
@END_Attrib
1 0 @F @F @F @F

@Var @RT(9)bInitDone @RT(0) @T @F @DT @RT(4)BOOL @RT(0) @T @T @BASIC 0 @F
@F @F
@T
@BEG_Attrib
3 @RT(0) @RT(0) @RT(0)
@END_Attrib
1 0 @F @F @F @F

@Var @RT(10)rCycleTime @RT(0) @T @F @DT @RT(4)REAL @RT(0) @T @T @BASIC 0 @F
@F @F
@T
@BEG_Attrib
3 @RT(0) @RT(0) @RT(0)
@END_Attrib
1 0 @F @F @F @F

@Var @RT(1)b @RT(0) @T @F @DT @RT(4)BOOL @RT(0) @T @T @BASIC 0 @F
@F @F
@T
@BEG_Attrib
3 @RT(0) @RT(0) @RT(0)
@END_Attrib
1 4 @F @F @F @F

@END_Dcl

@END_Export

@BEG_Export

@BEG_Algo
@POSTUPDATE_ALGORITHM @RT(17)pResetTotalEnergy @STRUCTURED_TEXT
@RT(0) @RT(18)sv_bResetTotEnergy @RT(7)TaskMid @F @F
@END_Algo

@BEG_Dcl
@RT(16)DclTreeContainer
0
@END_Dcl

@END_Export

@BEG_Export

@BEG_Algo
@PROCESS_ALGORITHM @RT(22)paInitDebugMeasurement @STRUCTURED_TEXT
@RT(0) @RT(0) @RT(8)TaskSlow @T @F
@END_Algo

@BEG_Dcl
@RT(16)DclTreeContainer
3
@Var @RT(6)fuName @RT(0) @T @F @DT @RT(11)STRING(255) @RT(0) @T @T @STRING 0 @F @RT(3)255 @F
@F @F
@T
@BEG_Attrib
3 @RT(0) @RT(0) @RT(0)
@END_Attrib
1 0 @F @F @F @F

@Var @RT(12)variableName @RT(0) @T @F @DT @RT(11)STRING(255) @RT(0) @T @T @STRING 0 @F @RT(3)255 @F
@F @F
@T
@BEG_Attrib
3 @RT(0) @RT(0) @RT(0)
@END_Attrib
1 0 @F @F @F @F

@Var @RT(8)swoState @RT(0) @T @T @DERIVED 0 @T @T @DT @RT(11)KSWO_Status @RT(0) @T @T @UNKNOWN 0 @F
@F @F
@T
@BEG_Attrib
3 @RT(0) @RT(0) @RT(0)
@END_Attrib
1 0 @F @F @F @F

@END_Dcl

@END_Export

@BEG_Export

@BEG_Algo
@POSTUPDATE_ALGORITHM @RT(11)pInitRecord @STRUCTURED_TEXT
@RT(0) @RT(16)sv_OperationMode @RT(10)TaskInject @F @F
@END_Algo

@BEG_Dcl
@RT(16)DclTreeContainer
0
@END_Dcl

@END_Export

@BEG_Export

@BEG_Algo
@POSTUPDATE_ALGORITHM @RT(14)pSampleMeasure @STRUCTURED_TEXT
@RT(0) @RT(22)sv_bStartSampleMeasure @RT(9)PU_Task_7 @F @F
@END_Algo

@BEG_Dcl
@RT(16)DclTreeContainer
0
@END_Dcl

@END_Export

@BEG_Export

@BEG_Algo
@PROCESS_ALGORITHM @RT(15)paSampleMeasure @STRUCTURED_TEXT
@RT(0) @RT(0) @RT(11)TaskHeating @F @F
@END_Algo

@BEG_Dcl
@RT(16)DclTreeContainer
5
@Var @RT(27)bLastMeasurementInitialized @RT(0) @T @T @RENAMED 0 @T @T @DT @RT(4)BOOL @RT(0) @T @T @BASIC 0 @F
@F @F
@T
@BEG_Attrib
3 @RT(0) @RT(0) @RT(0)
@END_Attrib
1 0 @F @F @F @F

@Var @RT(17)rMeasuredDuration @RT(0) @T @F @DT @RT(4)REAL @RT(0) @T @T @BASIC 0 @F
@F @F
@T
@BEG_Attrib
3 @RT(0) @RT(0) @RT(0)
@END_Attrib
1 0 @F @F @F @F

@Var @RT(10)dCycleTime @RT(0) @T @F @DT @RT(4)TIME @RT(0) @T @T @BASIC 0 @F
@F @F
@T
@BEG_Attrib
3 @RT(0) @RT(0) @RT(0)
@END_Attrib
1 0 @F @F @F @F

@Var @RT(10)rCycleTime @RT(0) @T @F @DT @RT(4)REAL @RT(0) @T @T @BASIC 0 @F
@F @F
@T
@BEG_Attrib
3 @RT(0) @RT(0) @RT(0)
@END_Attrib
1 0 @F @F @F @F

@Var @RT(12)rSetDuration @RT(0) @T @F @DT @RT(4)REAL @RT(0) @T @T @BASIC 0 @F
@F @F
@T
@BEG_Attrib
3 @RT(0) @RT(0) @RT(0)
@END_Attrib
1 0 @F @F @F @F

@END_Dcl

@END_Export

@BEG_Export

@BEG_Algo
@POSTUPDATE_ALGORITHM @RT(5)pInit @STRUCTURED_TEXT
@RT(0) @RT(12)sv_bInitDone @RT(9)PU_Task_7 @F @F
@END_Algo

@BEG_Dcl
@RT(16)DclTreeContainer
0
@END_Dcl

@END_Export

@BEG_Body
@TL(52)
(**************************************** WARNING ********************************************
 *** The KEBA Kemro K2 System including software is not intended for safety control tasks! ***
 ***                       For further information see Comment tab!                        ***
 *********************************************************************************************)

(*pointer to motor total power speedpump*)
mprMotorPowerSpeedpump := GET_SYNC_REFTO('Pump1.sv_rMotorTotalPower', T#0s, Status);

IF Status <> KSYS_Status_OK  THEN
   mprMotorPowerSpeedpump := GET_SYNC_REFTO('system.sv_rNull', T#0s, Status);
END_IF;

(*pointer to motor power elec.axes*)
mprMotorPowerEject := GET_SYNC_REFTO('Ejector1.sv_rMotorPowerEject', T#0s, Status);
IF Status <> KSYS_Status_OK  THEN
   mprMotorPowerEject := GET_SYNC_REFTO('system.sv_rNull', T#0s, Status);
END_IF;

mprMotorPowerInject:= GET_SYNC_REFTO('Injection1.sv_rMotorPowerInject', T#0s, Status);
IF Status <> KSYS_Status_OK  THEN
   mprMotorPowerInject := GET_SYNC_REFTO('system.sv_rNull', T#0s, Status);
END_IF;

mprMotorPowerPlast:= GET_SYNC_REFTO('Injection1.sv_rMotorPowerPlast', T#0s, Status);
IF Status <> KSYS_Status_OK  THEN
   mprMotorPowerPlast := GET_SYNC_REFTO('system.sv_rNull', T#0s, Status);
END_IF;

mprMotorPowerMold:= GET_SYNC_REFTO('Mold1.sv_rMotorPowerMold', T#0s, Status);
IF Status <> KSYS_Status_OK  THEN
   mprMotorPowerMold := GET_SYNC_REFTO('system.sv_rNull', T#0s, Status);
END_IF;

mprMotorPowerNozzle:= GET_SYNC_REFTO('Nozzle1.sv_rMotorPowerNozzle', T#0s, Status);
IF Status <> KSYS_Status_OK  THEN
   mprMotorPowerNozzle := GET_SYNC_REFTO('system.sv_rNull', T#0s, Status);
END_IF;

mprActCushion := GET_SYNC_REFTO('Injection1.sv_rCushion', T#0s, Status);
mprCushionZeroPosition := GET_SYNC_REFTO('Injection1.sv_rScrewZeroPosition', T#0s, Status);

mprHeatingPowerNozzle1 := GET_SYNC_REFTO('HeatingNozzle1.sv_rActHeatingPower', T#0s, Status);
IF Status = KSYS_Status_OK THEN
   mbHeatingPowerNozzle1Linked := TRUE;
END_IF;
mprHeatingPowerMold1 := GET_SYNC_REFTO('HeatingMold1.sv_rActHeatingPower', T#0s, Status);
IF Status = KSYS_Status_OK THEN
   mbHeatingPowerMold1Linked := TRUE;
END_IF;

STOP_PROCESS_ALGORITHM();

@END_Body

@@@BEG_Comment@@@
@TL(13)
@h    ! WARNING !
@h    The Kemro K2 system (including software) only meets category B according to EN 954-1,
@h    thus it is not intended for usage in safety-relevant control applications in the field
@h    of personal safety (e.g. emergency stop).
@h    To implement potentially necessary safety-relevant control tasks, always use additional
@h    external safety devices that are intended for the particular purpose, and meet the necessary
@h    functional safety.
@h    For further information see EN 954-1 (EN ISO 13849-1) and/or the K2-x00 user manual, chapter
@h    "CE conformity, directives and standards".

This algo initializes for the energy calculation

@@@END_Comment@@@

@BEG_Body
@TL(34)
(**************************************** WARNING ********************************************
 *** The KEBA Kemro K2 System including software is not intended for safety control tasks! ***
 ***                       For further information see Comment tab!                        ***
 *********************************************************************************************)

(*Calculation of the energy cosumption per shot*)
sv_rEnergyShot := mrActEnergy - mrTotEnergyLastShot;
mrTotEnergyLastShot := mrActEnergy;

(*Calculation of the energy cosumption per ccm*)
mrShotVolume := mprCushionZeroPosition^ - mprActCushion^;  (*calculate the shot volume*)

IF mrShotVolume <> 0.0 THEN
  sv_rEnergyShotVolume := sv_rEnergyShot / mrShotVolume;
ELSE
  sv_rEnergyShotVolume := 0.0;
END_IF;

//Synchronization to machine cycle
IF mbEnergyMeterLinked THEN
  IF sv_bStartSampleMeasure THEN

  //start the sample measurement
    IF NOT mbCycleRestarted THEN
      mbCycleRestarted := TRUE;
    END_IF;

    //shot counter for the sample measurement
    miShotCounter := miShotCounter + 1;
    END_IF;
END_IF;

@END_Body

@@@BEG_Comment@@@
@TL(12)
@h    ! WARNING !
@h    The Kemro K2 system (including software) only meets category B according to EN 954-1,
@h    thus it is not intended for usage in safety-relevant control applications in the field
@h    of personal safety (e.g. emergency stop).
@h    To implement potentially necessary safety-relevant control tasks, always use additional
@h    external safety devices that are intended for the particular purpose, and meet the necessary
@h    functional safety.
@h    For further information see EN 954-1 (EN ISO 13849-1) and/or the K2-x00 user manual, chapter
@h    "CE conformity, directives and standards".

This postupdate algorithms calculates the energy per shot and per ccm.

@@@END_Comment@@@

@BEG_Body
@TL(7)
(**************************************** WARNING ********************************************
 *** The KEBA Kemro K2 System including software is not intended for safety control tasks! ***
 ***                       For further information see Comment tab!                        ***
 *********************************************************************************************)
sv_rEnergyProduction := 0.0;             (*reset the energy per production*)
mrLastActEnergy := mrActEnergy;          (*copy the calculated energy of the last cycle*)

@END_Body

@@@BEG_Comment@@@
@TL(12)
@h    ! WARNING !
@h    The Kemro K2 system (including software) only meets category B according to EN 954-1,
@h    thus it is not intended for usage in safety-relevant control applications in the field
@h    of personal safety (e.g. emergency stop).
@h    To implement potentially necessary safety-relevant control tasks, always use additional
@h    external safety devices that are intended for the particular purpose, and meet the necessary
@h    functional safety.
@h    For further information see EN 954-1 (EN ISO 13849-1) and/or the K2-x00 user manual, chapter
@h    "CE conformity, directives and standards".

This AB calculates the energy per production.

@@@END_Comment@@@

@BEG_Body
@TL(17)
(**************************************** WARNING ********************************************
 *** The KEBA Kemro K2 System including software is not intended for safety control tasks! ***
 ***                       For further information see Comment tab!                        ***
 *********************************************************************************************)

(*Calculation of the energy cosumption per part*)
sv_rEnergyPart := mrActEnergy - mrTotEnergyLastPart;
mrTotEnergyLastPart := mrActEnergy;

(*Calculation of the energy cosumption in part mass*)
IF sv_rPartMass <> 0.0 THEN
    sv_rEnergyPartMass := sv_rEnergyPart / sv_rPartMass;
ELSE
    sv_rEnergyPartMass := 0.0;
END_IF;

@END_Body

@@@BEG_Comment@@@
@TL(11)
@h    ! WARNING !
@h    The Kemro K2 system (including software) only meets category B according to EN 954-1,
@h    thus it is not intended for usage in safety-relevant control applications in the field
@h    of personal safety (e.g. emergency stop).
@h    To implement potentially necessary safety-relevant control tasks, always use additional
@h    external safety devices that are intended for the particular purpose, and meet the necessary
@h    functional safety.
@h    For further information see EN 954-1 (EN ISO 13849-1) and/or the K2-x00 user manual, chapter
@h    "CE conformity, directives and standards".

This postupdate algorithm calculates the energy per gram.
@@@END_Comment@@@

@BEG_Body
@TL(71)
(**************************************** WARNING ********************************************
 *** The KEBA Kemro K2 System including software is not intended for safety control tasks! ***
 ***                       For further information see Comment tab!                        ***
 *********************************************************************************************)

(* Cycle time *)
IF NOT bInitDone THEN
   dCycleTime := GET_TASK_INTERVAL();
   rCycleTime := (LINT_TO_REAL(TIME_TO_LINT(dCycleTime))) / 1000000.0;
   bInitDone := TRUE;
END_IF;

(* Motor power estimated [kW] *)
mrMotorPower :=  mprMotorPowerSpeedpump^ +  mprMotorPowerEject^ +  mprMotorPowerInject^ +  mprMotorPowerPlast^ + mprMotorPowerMold^ + mprMotorPowerNozzle^;
b := WRITE_SVREAL_DIRECT(sv_rMotorPower, mrMotorPower);

(* Heat power estimated [W] *)
rHeatingPower := 0.0;
IF mbHeatingPowerNozzle1Linked THEN
   rHeatingPower := rHeatingPower + mprHeatingPowerNozzle1^;
END_IF;
IF mbHeatingPowerMold1Linked THEN
   rHeatingPower := rHeatingPower + mprHeatingPowerMold1^;
END_IF;
b := WRITE_SVREAL_DIRECT(sv_rHeatingPower, rHeatingPower);

(* Total power [kW] *)
IF mbEnergyMeterLinked THEN
   //Calculate the total power from measured total power
   b := WRITE_SVREAL_DIRECT(sv_rTotalPower, (sv_rMeasuredPower / 1000.0));
ELSE
   b := WRITE_SVREAL_DIRECT(sv_rTotalPower, (((rHeatingPower + sv_rIdlePower) / 1000.0 + mrMotorPower) / sv_rEfficiency));
END_IF;

(* Energy *)
IF mbEnergyMeterLinked THEN
   (* Total energy from power meter [kwh] *)
   sv_rTotalEnergy := (sv_rMeasuredEnergy - mrRecordedEnergy) / 1000.0; //measured value in Wh
   mrActEnergy := sv_rTotalEnergy;
   b := WRITE_SVREAL_DIRECT(sv_rMeasuredEnergyHMI, (sv_rMeasuredEnergy / 1000.0));

   (* Calculate the energy per production [kwh] *)
   IF sv_OperationMode >= nHalfAutomatic THEN
      b := WRITE_SVREAL_DIRECT(sv_rEnergyProduction, ((mrActEnergy - mrLastActEnergy) / 1000.0));
   END_IF;
ELSE
   (* Integration of power = Energy [kWs] *)
   mrActEnergy := mrTmpEnergy + sv_rTotalPower * rCycleTime;
   mrTmpEnergy := mrActEnergy;

   (* Calculate the energy per production [kwh] *)
   IF sv_OperationMode >= nHalfAutomatic THEN
      b := WRITE_SVREAL_DIRECT(sv_rEnergyProduction, ((mrActEnergy - mrLastActEnergy) / 3600.0));
   END_IF;

   (* Consumption of energy [kwh] *)
   sv_rTotalEnergy := (mrActEnergy / 3600.0 + mrRecordedEnergy);
END_IF;

(* Calibration *)
IF mbEnergyMeterLinked THEN
   (* Power calibration *)
   b := WRITE_SVREAL_DIRECT(sv_rTotalPowerCalibrated, ((sv_rMotorPower + (sv_rHeatingPower + sv_rIdlePower) / 1000.0) / sv_rEfficiency));

   (* Energy calibration *)
   mrActEnergyCalibrated := mrTmpEnergyCalibrated + sv_rTotalPowerCalibrated * rCycleTime;
   mrTmpEnergyCalibrated := mrActEnergyCalibrated;
   b := WRITE_SVREAL_DIRECT(sv_rTotalEnergyCalibrated, (mrActEnergyCalibrated / 3600.0));
END_IF;

@END_Body

@@@BEG_Comment@@@
@TL(11)
@h    ! WARNING !
@h    The Kemro K2 system (including software) only meets category B according to EN 954-1,
@h    thus it is not intended for usage in safety-relevant control applications in the field
@h    of personal safety (e.g. emergency stop).
@h    To implement potentially necessary safety-relevant control tasks, always use additional
@h    external safety devices that are intended for the particular purpose, and meet the necessary
@h    functional safety.
@h    For further information see EN 954-1 (EN ISO 13849-1) and/or the K2-x00 user manual, chapter
@h    "CE conformity, directives and standards".

This process algorithm calculates the energy.
@@@END_Comment@@@

@BEG_Body
@TL(31)
(**************************************** WARNING ********************************************
 *** The KEBA Kemro K2 System including software is not intended for safety control tasks! ***
 ***                       For further information see Comment tab!                        ***
 *********************************************************************************************)
(*reset the energy calculator*)
IF sv_bResetTotEnergy THEN
   //when power meter is used, record the last measured total energy,
   //and calculate always the difference between the actual measured value and recorded value
   //when estimation is used, integration of power with initial value 0 would be restarted
   IF mbEnergyMeterLinked THEN
     mrRecordedEnergy := sv_rMeasuredEnergy;
   ELSE
     mrRecordedEnergy := 0.0;
   END_IF;

   mrActEnergy := 0.0;
   mrTmpEnergy := 0.0;
   sv_rTotalEnergy := 0.0;
   mrLastActEnergy := 0.0;
   mrTotEnergyLastShot := 0.0;
   mrTotEnergyLastPart := 0.0;
   sv_bResetTotEnergy := FALSE;

   //calibration
   IF mbEnergyMeterLinked THEN
     mrActEnergyCalibrated := 0.0;
     mrTmpEnergyCalibrated := 0.0;
     sv_rTotalEnergyCalibrated := 0.0;
   END_IF;
END_IF;

@END_Body

@@@BEG_Comment@@@
@TL(11)
@h    ! WARNING !
@h    The Kemro K2 system (including software) only meets category B according to EN 954-1,
@h    thus it is not intended for usage in safety-relevant control applications in the field
@h    of personal safety (e.g. emergency stop).
@h    To implement potentially necessary safety-relevant control tasks, always use additional
@h    external safety devices that are intended for the particular purpose, and meet the necessary
@h    functional safety.
@h    For further information see EN 954-1 (EN ISO 13849-1) and/or the K2-x00 user manual, chapter
@h    "CE conformity, directives and standards".

This postupdate algorithm resets the energy calculation.
@@@END_Comment@@@

@BEG_Body
@TL(24)
(**************************************** WARNING ********************************************
 *** The KEBA Kemro K2 System including software is not intended for safety control tasks! ***
 ***                       For further information see Comment tab!                        ***
 *********************************************************************************************)
fuName := GET_MY_FU_NAME();
variableName := CONCAT(fuName,'.rMotorPowerCalc kW');
swoState := KSWO_AddVariable( Task := TaskInject,
                              Name := variableName,
                              Variable := sv_rMotorPower);
variableName := CONCAT(fuName,'.rTotalEnergyMeasured kWh');
swoState := KSWO_AddVariable( Task := TaskInject,
                              Name := variableName,
                              Variable := sv_rTotalEnergy);
variableName := CONCAT(fuName,'.rTotalEnergyCalibrated kWh');
swoState := KSWO_AddVariable( Task := TaskInject,
                              Name := variableName,
                              Variable := sv_rTotalEnergyCalibrated);
variableName := CONCAT(fuName,'.rTotalPower kW');
swoState := KSWO_AddVariable( Task := TaskInject,
                              Name := variableName,
                              Variable := sv_rTotalPower);
STOP_PROCESS_ALGORITHM();

@END_Body

@@@BEG_Comment@@@
@TL(0)

@@@END_Comment@@@

@BEG_Body
@TL(10)
(**************************************** WARNING ********************************************
 *** The KEBA Kemro K2 System including software is not intended for safety control tasks! ***
 ***                       For further information see Comment tab!                        ***
 *********************************************************************************************)
(*Reset the last sum*)
IF sv_OperationMode = nFullAutomatic THEN
    mrTotEnergyLastShot := 0.0;
    mrTotEnergyLastPart := 0.0;
END_IF;

@END_Body

@@@BEG_Comment@@@
@TL(12)
@h    ! WARNING !
@h    The Kemro K2 system (including software) only meets category B according to EN 954-1,
@h    thus it is not intended for usage in safety-relevant control applications in the field
@h    of personal safety (e.g. emergency stop).
@h    To implement potentially necessary safety-relevant control tasks, always use additional
@h    external safety devices that are intended for the particular purpose, and meet the necessary
@h    functional safety.
@h    For further information see EN 954-1 (EN ISO 13849-1) and/or the K2-x00 user manual, chapter
@h    "CE conformity, directives and standards".

This postppdate algorithm resets the temp variables for sum.

@@@END_Comment@@@

@BEG_Body
@TL(5)
//start the sample measurement
IF sv_bStartSampleMeasure THEN
  START_PROCESS_ALGORITHM(paSampleMeasure);
END_IF;

@END_Body

@@@BEG_Comment@@@
@TL(0)

@@@END_Comment@@@

@BEG_Body
@TL(35)
IF mbCycleRestarted THEN

  //Initialization of measurement
  IF NOT bLastMeasurementInitialized THEN
    bLastMeasurementInitialized := TRUE;
    mrRecordedSampleEnergy := sv_rMeasuredEnergy;  //read the latest measured energy
    miShotCounter := 0;                         //reset the shotcounter for sampling
    rMeasuredDuration := 0.0;                   //reset the duration for sampling
    dCycleTime := GET_TASK_INTERVAL();
    rCycleTime := (LINT_TO_REAL(TIME_TO_LINT(dCycleTime))) / 1.0e6;  //in seconds
    rSetDuration := LINT_TO_REAL(TIME_TO_LINT(sv_dSetDuration)) / 1.0e6;   //set duration in seconds
  END_IF;

  //Energy consumption from starting the sampling
  sv_rSampleMeasuredEnergy := (sv_rMeasuredEnergy - mrRecordedSampleEnergy) / 1.0e3;

  rMeasuredDuration := rMeasuredDuration + rCycleTime;
  sv_dMeasuredDuration := LINT_TO_TIME(REAL_TO_LINT(rMeasuredDuration * 1.0e6));    //in mins

  //Auto-Stop dependant on shot counter and set measurement duration
  //Automatically stopped when shot counter or duration first is reached
  IF ((miShotCounter >= sv_iAutoStopShotCounter) AND (sv_iAutoStopShotCounter <> 0))
                             OR ((rMeasuredDuration >= rSetDuration) AND (rSetDuration <> 0.0)) OR (NOT sv_bStartSampleMeasure) THEN

      mbCycleRestarted := FALSE;
    sv_bStartSampleMeasure := FALSE;
    bLastMeasurementInitialized := FALSE;

    STOP_PROCESS_ALGORITHM();
  END_IF;
ELSE  //waiting for the start of next cycle
  sv_rSampleMeasuredEnergy := 0.0; //reset the measurement
  sv_dMeasuredDuration := t#0s;    //reset the timer
END_IF;

@END_Body

@@@BEG_Comment@@@
@TL(0)

@@@END_Comment@@@

@BEG_Body
@TL(16)
//Energy meter is linked
IF sv_NumberOfDevices[cCompEnergyMeter] <> 0 THEN
  mbEnergyMeterLinked := TRUE;
END_IF;

// Calculate/Measure power/energy cyclically
START_PROCESS_ALGORITHM(paCalcAndMeasure);

IF NOT mbEnergyMeterLinked THEN
  mrRecordedEnergy := sv_rTotalEnergy;
ELSE
  mrRecordedEnergy := sv_rMeasuredEnergy; //initialization
END_IF;

@END_Body

@@@BEG_Comment@@@
@TL(0)

@@@END_Comment@@@
@END_Body

@END_Contents

(* ---- ABInfoLog.pu ---- *)
(*
@h    ! WARNING !
@h    The Kemro K2 system (including software) only meets category B according to EN 954-1,
@h    thus it is not intended for usage in safety-relevant control applications in the field
@h    of personal safety (e.g. emergency stop).
@h    To implement potentially necessary safety-relevant control tasks, always use additional
@h    external safety devices that are intended for the particular purpose, and meet the necessary
@h    functional safety.
@h    For further information see EN 954-1 (EN ISO 13849-1) and/or the K2-x00 user manual, chapter
@h    "CE conformity, directives and standards".

This algorithm block reacts on changes of infolog relevant machine states and creates an infolog entry
in group --- IlogUser0 ---.
*)

IMPORT_OVER_LISTFILE
 KPROT_UserInfoLog
, KPROT_Status

END_IMPORT

ALGORITHM_BLOCK ABInfoLog #DUMMY_EDIT_BLOCK

SYSTEM_VAR
 sv_bAllMotorsRunning : BOOL;
 sv_bMoldHeatingOn : BOOL;
 sv_bNozzleHeatingOn : BOOL;
END_VAR

SYSTEM_OBJECT
 PU_Task_13 : TASK;
END_OBJECT

VAR
 mStatus : KPROT_Status;
END_VAR

POSTUPDATE_ALGORITHM pLogMotorOnOff ON PU_Task_13 WITH sv_bAllMotorsRunning

VAR_IN_OUT
 bOn : BOOL;
END_VAR
#BEGIN_EDIT_BLOCK
(**************************************** WARNING ********************************************
 *** The KEBA Kemro K2 System including software is not intended for safety control tasks! ***
 ***                       For further information see Comment tab!                        ***
 *********************************************************************************************)

IF (bOn) THEN
  mStatus := KPROT_UserInfoLog("%5s", 0, 0, 0, 0, "Motor on");
ELSE
  mStatus := KPROT_UserInfoLog("%5s", 0, 0, 0, 0, "Motor off");
END_IF;

;#END_EDIT_BLOCK END_ALGORITHM

POSTUPDATE_ALGORITHM pLogMoldHeatingOnOff ON PU_Task_13 WITH sv_bMoldHeatingOn

VAR_IN_OUT
 bOn : BOOL;
END_VAR
#BEGIN_EDIT_BLOCK
(**************************************** WARNING ********************************************
 *** The KEBA Kemro K2 System including software is not intended for safety control tasks! ***
 ***                       For further information see Comment tab!                        ***
 *********************************************************************************************)

IF (bOn) THEN
  mStatus := KPROT_UserInfoLog("%5s", 0, 0, 0, 0, "Mold heating on");
ELSE
  mStatus := KPROT_UserInfoLog("%5s", 0, 0, 0, 0, "Mold heating off");
END_IF;

;#END_EDIT_BLOCK END_ALGORITHM

POSTUPDATE_ALGORITHM pLogNozzleHeatingOnOff ON PU_Task_13 WITH sv_bNozzleHeatingOn

VAR_IN_OUT
 bOn : BOOL;
END_VAR
#BEGIN_EDIT_BLOCK
(**************************************** WARNING ********************************************
 *** The KEBA Kemro K2 System including software is not intended for safety control tasks! ***
 ***                       For further information see Comment tab!                        ***
 *********************************************************************************************)

IF (bOn) THEN
  mStatus := KPROT_UserInfoLog("%5s", 0, 0, 0, 0, "Nozzle heating on");
ELSE
  mStatus := KPROT_UserInfoLog("%5s", 0, 0, 0, 0, "Nozzle heating off");
END_IF;

;#END_EDIT_BLOCK END_ALGORITHM

END_ALGORITHM_BLOCK

#END_OF_IEC_PART

@Puma @IecEditor 6 131 @Pou 25
@@@BEG_Comment@@@
@h    ! WARNING !
@h    The Kemro K2 system (including software) only meets category B according to EN 954-1,
@h    thus it is not intended for usage in safety-relevant control applications in the field
@h    of personal safety (e.g. emergency stop).
@h    To implement potentially necessary safety-relevant control tasks, always use additional
@h    external safety devices that are intended for the particular purpose, and meet the necessary
@h    functional safety.
@h    For further information see EN 954-1 (EN ISO 13849-1) and/or the K2-x00 user manual, chapter
@h    "CE conformity, directives and standards".

This algorithm block reacts on changes of infolog relevant machine states and creates an infolog entry
in group --- IlogUser0 ---.
@@@END_Comment@@@

@BEG_Contents

@BEG_Func
@RT(17)FuncTreeContainer
1
@Var @RT(17)KPROT_UserInfoLog @RT(0) @T @T @DERIVED 0 @F @RT(37)KEBA_STANDARD_FUNCTION : KPROT_Status @F
@T
@BEG_Attrib
0 @RT(0) @RT(0)
@END_Attrib
1 1 @F @F @F @F

@END_Func

@BEG_Const
@RT(18)ConstTreeContainer
0
@END_Const

@BEG_Export

@BEG_Kind
@ALGORITHM_BLOCK @RT(9)ABInfoLog @STRUCTURED_TEXT
@RT(0) @RT(0) @RT(0)
@END_Kind

@BEG_Dcl
@RT(16)DclTreeContainer
5
@Var @RT(10)PU_Task_13 @RT(0) @T @F @DT @RT(4)TASK @RT(0) @T @T @BASIC 0 @F
@F @F
@T
@BEG_Attrib
3 @RT(0) @RT(0) @RT(0)
@END_Attrib
1 7 @F @F @F @F

@Var @RT(20)sv_bAllMotorsRunning @RT(0) @T @F @DT @RT(4)BOOL @RT(0) @T @T @BASIC 0 @F
@F @F
@T
@BEG_Attrib
3 @RT(0) @RT(0) @RT(0)
@END_Attrib
1 8 @F @F @F @F

@Var @RT(17)sv_bMoldHeatingOn @RT(0) @T @F @DT @RT(4)BOOL @RT(0) @T @T @BASIC 0 @F
@F @F
@T
@BEG_Attrib
3 @RT(0) @RT(0) @RT(0)
@END_Attrib
1 8 @F @F @F @F

@Var @RT(19)sv_bNozzleHeatingOn @RT(0) @T @F @DT @RT(4)BOOL @RT(0) @T @T @BASIC 0 @F
@F @F
@T
@BEG_Attrib
3 @RT(0) @RT(0) @RT(0)
@END_Attrib
1 8 @F @F @F @F

@Var @RT(7)mStatus @RT(0) @T @T @DERIVED 0 @F @RT(12)KPROT_Status @F
@T
@BEG_Attrib
3 @RT(0) @RT(0) @RT(0)
@END_Attrib
1 0 @F @F @F @F

@END_Dcl

@END_Export

@BEG_Body

3

@BEG_Export

@BEG_Algo
@POSTUPDATE_ALGORITHM @RT(14)pLogMotorOnOff @STRUCTURED_TEXT
@RT(0) @RT(20)sv_bAllMotorsRunning @RT(10)PU_Task_13 @F @F
@END_Algo

@BEG_Dcl
@RT(16)DclTreeContainer
1
@Var @RT(3)bOn @RT(0) @T @F @DT @RT(4)BOOL @RT(0) @T @T @BASIC 0 @F
@F @F
@T
@BEG_Attrib
3 @RT(0) @RT(0) @RT(0)
@END_Attrib
1 2 @F @F @F @F

@END_Dcl

@END_Export

@BEG_Export

@BEG_Algo
@POSTUPDATE_ALGORITHM @RT(20)pLogMoldHeatingOnOff @STRUCTURED_TEXT
@RT(0) @RT(17)sv_bMoldHeatingOn @RT(10)PU_Task_13 @F @F
@END_Algo

@BEG_Dcl
@RT(16)DclTreeContainer
1
@Var @RT(3)bOn @RT(0) @T @F @DT @RT(4)BOOL @RT(0) @T @T @BASIC 0 @F
@F @F
@T
@BEG_Attrib
3 @RT(0) @RT(0) @RT(0)
@END_Attrib
1 2 @F @F @F @F

@END_Dcl

@END_Export

@BEG_Export

@BEG_Algo
@POSTUPDATE_ALGORITHM @RT(22)pLogNozzleHeatingOnOff @STRUCTURED_TEXT
@RT(0) @RT(19)sv_bNozzleHeatingOn @RT(10)PU_Task_13 @F @F
@END_Algo

@BEG_Dcl
@RT(16)DclTreeContainer
1
@Var @RT(3)bOn @RT(0) @T @F @DT @RT(4)BOOL @RT(0) @T @T @BASIC 0 @F
@F @F
@T
@BEG_Attrib
3 @RT(0) @RT(0) @RT(0)
@END_Attrib
1 2 @F @F @F @F

@END_Dcl

@END_Export

@BEG_Body
@TL(11)
(**************************************** WARNING ********************************************
 *** The KEBA Kemro K2 System including software is not intended for safety control tasks! ***
 ***                       For further information see Comment tab!                        ***
 *********************************************************************************************)

IF (bOn) THEN
  mStatus := KPROT_UserInfoLog("%5s", 0, 0, 0, 0, "Motor on");
ELSE
  mStatus := KPROT_UserInfoLog("%5s", 0, 0, 0, 0, "Motor off");
END_IF;

@END_Body

@@@BEG_Comment@@@
@TL(0)

@@@END_Comment@@@

@BEG_Body
@TL(11)
(**************************************** WARNING ********************************************
 *** The KEBA Kemro K2 System including software is not intended for safety control tasks! ***
 ***                       For further information see Comment tab!                        ***
 *********************************************************************************************)

IF (bOn) THEN
  mStatus := KPROT_UserInfoLog("%5s", 0, 0, 0, 0, "Mold heating on");
ELSE
  mStatus := KPROT_UserInfoLog("%5s", 0, 0, 0, 0, "Mold heating off");
END_IF;

@END_Body

@@@BEG_Comment@@@
@TL(0)

@@@END_Comment@@@

@BEG_Body
@TL(11)
(**************************************** WARNING ********************************************
 *** The KEBA Kemro K2 System including software is not intended for safety control tasks! ***
 ***                       For further information see Comment tab!                        ***
 *********************************************************************************************)

IF (bOn) THEN
  mStatus := KPROT_UserInfoLog("%5s", 0, 0, 0, 0, "Nozzle heating on");
ELSE
  mStatus := KPROT_UserInfoLog("%5s", 0, 0, 0, 0, "Nozzle heating off");
END_IF;

@END_Body

@@@BEG_Comment@@@
@TL(0)

@@@END_Comment@@@
@END_Body

@END_Contents

(* ---- ABPanelButtonRegister.pu ---- *)
IMPORT_OVER_LISTFILE
 GET_TASK_INTERVAL
, tevPanelButtonRegister
, tyPanelButton
, tsTraceLevel
, tevPanelButtonRegisterData
, tsPanelButton

END_IMPORT

ALGORITHM_BLOCK ABPanelButtonRegister #DUMMY_EDIT_BLOCK

SYSTEM_VAR
 sv_PanelButtons : tyPanelButton;
 sv_iPanelButtonCnt : DINT;
 sv_bUsePanelHeartbeat : BOOL;
 sv_iPanelHeartbeat : DINT;
 sv_iPanelMovementSelector : DINT;
 sv_iPanelHeartbeatInterval : DINT;
 sv_iPanelHeartbeatTolerance : DINT;
 sv_TraceLevel : tsTraceLevel;
 sv_bInitDone : BOOL;
END_VAR

SYSTEM_OBJECT
 evPanelButtonRegister : tevPanelButtonRegister;
 EV_Task_3 : TASK;
 PU_Task_3 : TASK;
 PU_Task_7 : TASK;
 TaskMid : TASK;
END_OBJECT

VAR
 miAliveTicks : DINT (* Cycles to check alive flag *);
 mpbActionVar1 : REFTO BOOL;
 mpbActionVar2 : REFTO BOOL;
END_VAR

(*
get instance data if start event is received

attention:
taskslot is asigned to make sure that execution is done before evaStart in ABControl.pu
*)

EVENT_ALGORITHM evaRegisterPanelButton ON EV_Task_3(50) WITH evPanelButtonRegister

VAR_INPUT
 EventData : tevPanelButtonRegisterData;
END_VAR

VAR
 dummy : DINT;
 sText : STRING(255);
END_VAR
#BEGIN_EDIT_BLOCK
(**************************************** WARNING ********************************************
 *** The KEBA Kemro K2 System including software is not intended for safety control tasks! ***
 ***                       For further information see Comment tab!                        ***
 *********************************************************************************************)

IF sv_iPanelButtonCnt >= cMaxPanelButtons THEN
    IF sv_TraceLevel.bApplication THEN
       sText := CONCAT('ABPanelButtonRegister: number of panel buttons exceeded maximum, omitting button from component %d/%d',
                   DINT_TO_STRING(EventData.Button.iCompId), DINT_TO_STRING(EventData.Button.iIndexId));
       dummy := Print(sText);
    END_IF;
    RETURN;
END_IF;
// This array contains all possible movements/actions that can be used within an HMI application.
// The HMI can read this array in order to dynamically create a HMI machine operation panel on
// the visualisation system.
sv_iPanelButtonCnt := sv_iPanelButtonCnt + 1;
sv_PanelButtons[sv_iPanelButtonCnt] := EventData.Button;

;#END_EDIT_BLOCK END_ALGORITHM

POSTUPDATE_ALGORITHM pMoveSelectorChanged ON PU_Task_7 WITH sv_iPanelMovementSelector

VAR
 Button : tsPanelButton;
END_VAR
#BEGIN_EDIT_BLOCK
(**************************************** WARNING ********************************************
 *** The KEBA Kemro K2 System including software is not intended for safety control tasks! ***
 ***                       For further information see Comment tab!                        ***
 *********************************************************************************************)

IF (sv_iPanelMovementSelector > 0) THEN
   Button := sv_PanelButtons[sv_iPanelMovementSelector];
   mpbActionVar1 := Button.pbActionVar1;
   mpbActionVar2 := Button.pbActionVar2;
ELSE
   mpbActionVar1 := EMPTY;
   mpbActionVar2 := EMPTY;
END_IF;

;#END_EDIT_BLOCK END_ALGORITHM

PROCESS_ALGORITHM paCheckHeartbeat ON TaskMid

VAR
 bTimeout : BOOL;
 bOutputActive : BOOL;
 iHeartbeat : DINT;
 bAlive : BOOL;
 iCnt : DINT;
 dummy : DINT;
 sText : STRING(255);
END_VAR

(* IecGraph-Code *)

(* init step *)
INITIAL_STEP S_Idle:
Action1 (P);
Output_Active (N);
END_STEP

ACTION Action1: #BEGIN_EDIT_BLOCK
bTimeout := FALSE

;#END_EDIT_BLOCK END_ACTION (*Action1*)
ACTION Output_Active: #BEGIN_EDIT_BLOCK
IF (mpbActionVar1 = EMPTY OR mpbActionVar2 = EMPTY) THEN
   bOutputActive := FALSE;
ELSE
   bOutputActive := mpbActionVar1^ = TRUE OR mpbActionVar2^ = TRUE;
END_IF;

;#END_EDIT_BLOCK END_ACTION (*Output_Active*)

(* steps *)
STEP S_OutputActive:
Action2 (P);
Check_Heartbeat (N);
END_STEP

ACTION Action2: #BEGIN_EDIT_BLOCK
iHeartbeat := sv_iPanelHeartbeat;
bAlive := TRUE;
iCnt := 0;

;#END_EDIT_BLOCK END_ACTION (*Action2*)
ACTION Check_Heartbeat: #BEGIN_EDIT_BLOCK
IF (mpbActionVar1 = EMPTY AND mpbActionVar2 = EMPTY) THEN
   bOutputActive := FALSE;
ELSE
   bOutputActive := FALSE;
   IF (mpbActionVar1 <> EMPTY) THEN
      bOutputActive := mpbActionVar1^;
   END_IF;
   IF (NOT bOutputActive AND mpbActionVar2 <> EMPTY) THEN
      bOutputActive := mpbActionVar2^;
   END_IF;

   IF (sv_iPanelHeartbeat <> iHeartbeat) THEN
      (* heartbeat counter changed while output active *)
      bAlive := TRUE;
      iHeartbeat := sv_iPanelHeartbeat;
      iCnt := 0;
   ELSE
      iCnt := iCnt + 1;
      IF iCnt > miAliveTicks THEN
         bAlive := FALSE;
      END_IF;
   END_IF;
END_IF;

;#END_EDIT_BLOCK END_ACTION (*Check_Heartbeat*)
STEP S_Timeout:
Reset_IO (N);
END_STEP

ACTION Reset_IO: #BEGIN_EDIT_BLOCK
(* Safety reset *)
IF (mpbActionVar1 <> EMPTY) THEN
   mpbActionVar1^ := FALSE;
END_IF;
IF (mpbActionVar2 <> EMPTY) THEN
   mpbActionVar2^ := FALSE;
END_IF;
IF sv_TraceLevel.bApplication THEN
   sText := CONCAT('HMI timeout, output was reset by heartbeat detection, ticks detected ',
                        DINT_TO_STRING(iCnt),
                        ', maximum ',
                        DINT_TO_STRING(miAliveTicks));
   dummy := Print(sText);
END_IF;

;#END_EDIT_BLOCK END_ACTION (*Reset_IO*)

(* transitions *)
TRANSITION Trans1 (* Trans1 *) FROM S_Idle TO S_OutputActive :=  #BEGIN_EDIT_BLOCK
bOutputActive = TRUE

;#END_EDIT_BLOCK
END_TRANSITION

TRANSITION Trans3 (* Trans3 *) FROM S_OutputActive TO S_Idle :=  #BEGIN_EDIT_BLOCK
NOT bOutputActive
;#END_EDIT_BLOCK
END_TRANSITION

TRANSITION HMI_Disconnected (* Trans2 *) FROM S_OutputActive TO S_Timeout :=  #BEGIN_EDIT_BLOCK
bAlive = FALSE
;#END_EDIT_BLOCK
END_TRANSITION

TRANSITION Trans4 (* Trans4 *) FROM S_Timeout TO S_Idle :=  #BEGIN_EDIT_BLOCK
TRUE
;#END_EDIT_BLOCK
END_TRANSITION

(* end IecGraph-Code *)
(* sfc-code *)

(* stand alone actions *)
// ACTION Action3: #BEGIN_EDIT_BLOCK

// ;#END_EDIT_BLOCK END_ACTION (*Action3*)
(* end sfc-code *)

END_ALGORITHM

ALGORITHM aSetHeartbeatInterval

VAR
 iInterval : DINT;
END_VAR
#BEGIN_EDIT_BLOCK
(* Currently checked in TaskMid *)
iInterval := LINT_TO_DINT(TIME_TO_LINT(GET_TASK_INTERVAL(TaskMid))/1000);

IF sv_iPanelHeartbeatInterval < iInterval THEN
   sv_iPanelHeartbeatInterval := iInterval;
END_IF;

miAliveTicks := (sv_iPanelHeartbeatInterval + sv_iPanelHeartbeatTolerance)/(iInterval);

;#END_EDIT_BLOCK END_ALGORITHM

POSTUPDATE_ALGORITHM pHeartbeatInterval ON PU_Task_7 WITH sv_iPanelHeartbeatInterval, sv_iPanelHeartbeatTolerance

#BEGIN_EDIT_BLOCK

aSetHeartbeatInterval();

;#END_EDIT_BLOCK END_ALGORITHM

POSTUPDATE_ALGORITHM pInit ON PU_Task_3 WITH sv_bInitDone, sv_bUsePanelHeartbeat

#BEGIN_EDIT_BLOCK

aSetHeartbeatInterval();
IF (sv_bUsePanelHeartbeat) THEN
   START_PROCESS_ALGORITHM(paCheckHeartbeat);
ELSE
   STOP_PROCESS_ALGORITHM(paCheckHeartbeat);
END_IF;

;#END_EDIT_BLOCK END_ALGORITHM

END_ALGORITHM_BLOCK

#END_OF_IEC_PART

@Puma @IecEditor 6 150 @Pou 25
@@@BEG_Comment@@@

@@@END_Comment@@@

@BEG_Contents

@BEG_Func
@RT(17)FuncTreeContainer
1
@Var @RT(17)GET_TASK_INTERVAL @RT(0) @T @T @DERIVED 0 @F @RT(22)KEBA_STANDARD_FUNCTION @F
@T
@BEG_Attrib
0 @RT(0) @RT(0)
@END_Attrib
1 1 @F @F @F @F

@END_Func

@BEG_Const
@RT(18)ConstTreeContainer
0
@END_Const

@BEG_Export

@BEG_Kind
@ALGORITHM_BLOCK @RT(21)ABPanelButtonRegister @STRUCTURED_TEXT
@RT(0) @RT(0) @RT(0)
@END_Kind

@BEG_Dcl
@RT(16)DclTreeContainer
17
@Var @RT(21)evPanelButtonRegister @RT(0) @T @T @DERIVED 0 @T @T @DT @RT(22)tevPanelButtonRegister @RT(0) @T @T @UNKNOWN 0 @F
@F @F
@T
@BEG_Attrib
3 @RT(0) @RT(0) @RT(0)
@END_Attrib
1 7 @F @F @F @F

@Var @RT(15)sv_PanelButtons @RT(0) @T @T @DERIVED 0 @T @T @DT @RT(13)tyPanelButton @RT(0) @T @T @UNKNOWN 0 @F
@F @F
@T
@BEG_Attrib
3 @RT(0) @RT(0) @RT(0)
@END_Attrib
1 8 @F @F @F @F

@Var @RT(18)sv_iPanelButtonCnt @RT(0) @T @F @DT @RT(4)DINT @RT(0) @T @T @BASIC 0 @F
@F @F
@T
@BEG_Attrib
3 @RT(0) @RT(0) @RT(0)
@END_Attrib
1 8 @F @F @F @F

@Var @RT(9)EV_Task_3 @RT(0) @T @F @DT @RT(4)TASK @RT(0) @T @T @BASIC 0 @F
@F @F
@T
@BEG_Attrib
3 @RT(0) @RT(0) @RT(0)
@END_Attrib
1 7 @F @F @F @F

@Var @RT(9)PU_Task_3 @RT(0) @T @F @DT @RT(4)TASK @RT(0) @T @T @BASIC 0 @F
@F @F
@T
@BEG_Attrib
3 @RT(0) @RT(0) @RT(0)
@END_Attrib
1 7 @F @F @F @F

@Var @RT(9)PU_Task_7 @RT(0) @T @F @DT @RT(4)TASK @RT(0) @T @T @BASIC 0 @F
@F @F
@T
@BEG_Attrib
3 @RT(0) @RT(0) @RT(0)
@END_Attrib
1 7 @F @F @F @F

@Var @RT(7)TaskMid @RT(0) @T @F @DT @RT(4)TASK @RT(0) @T @T @BASIC 0 @F
@F @F
@T
@BEG_Attrib
3 @RT(0) @RT(0) @RT(0)
@END_Attrib
1 7 @F @F @F @F

@Var @RT(21)sv_bUsePanelHeartbeat @RT(0) @T @F @DT @RT(4)BOOL @RT(0) @T @T @BASIC 0 @F
@F @F
@T
@BEG_Attrib
3 @RT(0) @RT(0) @RT(0)
@END_Attrib
1 8 @F @F @F @F

@Var @RT(18)sv_iPanelHeartbeat @RT(0) @T @F @DT @RT(4)DINT @RT(0) @T @T @BASIC 0 @F
@F @F
@T
@BEG_Attrib
3 @RT(0) @RT(0) @RT(0)
@END_Attrib
1 8 @F @F @F @F

@Var @RT(25)sv_iPanelMovementSelector @RT(0) @T @F @DT @RT(4)DINT @RT(0) @T @T @BASIC 0 @F
@F @F
@T
@BEG_Attrib
3 @RT(0) @RT(0) @RT(0)
@END_Attrib
1 8 @F @F @F @F

@Var @RT(26)sv_iPanelHeartbeatInterval @RT(0) @T @F @DT @RT(4)DINT @RT(0) @T @T @BASIC 0 @F
@F @F
@T
@BEG_Attrib
3 @RT(0) @RT(0) @RT(0)
@END_Attrib
1 8 @F @F @F @F

@Var @RT(27)sv_iPanelHeartbeatTolerance @RT(0) @T @F @DT @RT(4)DINT @RT(0) @T @T @BASIC 0 @F
@F @F
@T
@BEG_Attrib
3 @RT(0) @RT(0) @RT(0)
@END_Attrib
1 8 @F @F @F @F

@Var @RT(13)sv_TraceLevel @RT(0) @T @T @DERIVED 0 @F @RT(12)tsTraceLevel @F
@T
@BEG_Attrib
3 @RT(0) @RT(0) @RT(0)
@END_Attrib
1 8 @F @F @F @F

@Var @RT(12)sv_bInitDone @RT(0) @T @F @DT @RT(4)BOOL @RT(0) @T @T @BASIC 0 @F
@F @F
@T
@BEG_Attrib
3 @RT(0) @RT(0) @RT(0)
@END_Attrib
1 8 @F @F @F @F

@Var @RT(12)miAliveTicks @RT(0) @T @F @DT @RT(4)DINT @RT(0) @T @T @BASIC 0 @F
@F @F
@T
@BEG_Attrib
3 @RT(0) @RT(26)Cycles to check alive flag @RT(0)
@END_Attrib
1 0 @F @F @F @F

@Var @RT(13)mpbActionVar1 @RT(0) @T @T @REFTO 0 @T @DT @RT(4)BOOL @RT(0) @T @T @BASIC 0 @F
@F @F
@T
@BEG_Attrib
3 @RT(0) @RT(0) @RT(0)
@END_Attrib
1 0 @F @F @F @F

@Var @RT(13)mpbActionVar2 @RT(0) @T @T @REFTO 0 @T @DT @RT(4)BOOL @RT(0) @T @T @BASIC 0 @F
@F @F
@T
@BEG_Attrib
3 @RT(0) @RT(0) @RT(0)
@END_Attrib
1 0 @F @F @F @F

@END_Dcl

@END_Export

@BEG_Body

6

@BEG_Export

@BEG_Algo
@EVENT_ALGORITHM @RT(22)evaRegisterPanelButton @STRUCTURED_TEXT
@RT(0) @RT(21)evPanelButtonRegister @RT(13)EV_Task_3(50) @F @F
@END_Algo

@BEG_Dcl
@RT(16)DclTreeContainer
3
@Var @RT(9)EventData @RT(0) @T @T @DERIVED 0 @T @T @DT @RT(26)tevPanelButtonRegisterData @RT(0) @T @T @UNKNOWN 0 @F
@F @F
@T
@BEG_Attrib
3 @RT(0) @RT(0) @RT(0)
@END_Attrib
1 1 @F @F @F @F

@Var @RT(5)dummy @RT(0) @T @F @DT @RT(4)DINT @RT(0) @T @T @BASIC 0 @F
@F @F
@T
@BEG_Attrib
3 @RT(0) @RT(0) @RT(0)
@END_Attrib
1 0 @F @F @F @F

@Var @RT(5)sText @RT(0) @T @F @DT @RT(11)STRING(255) @RT(0) @T @T @STRING 0 @F @RT(3)255 @F
@F @F
@T
@BEG_Attrib
3 @RT(0) @RT(0) @RT(0)
@END_Attrib
1 0 @F @F @F @F

@END_Dcl

@END_Export

@BEG_Export

@BEG_Algo
@POSTUPDATE_ALGORITHM @RT(20)pMoveSelectorChanged @STRUCTURED_TEXT
@RT(0) @RT(25)sv_iPanelMovementSelector @RT(9)PU_Task_7 @F @F
@END_Algo

@BEG_Dcl
@RT(16)DclTreeContainer
1
@Var @RT(6)Button @RT(0) @T @T @DERIVED 0 @T @T @DT @RT(13)tsPanelButton @RT(0) @T @T @UNKNOWN 0 @F
@F @F
@T
@BEG_Attrib
3 @RT(0) @RT(0) @RT(0)
@END_Attrib
1 0 @F @F @F @F

@END_Dcl

@END_Export

@BEG_Export

@BEG_Algo
@PROCESS_ALGORITHM @RT(16)paCheckHeartbeat @SEQUENTIAL_FLOW_CHART
@RT(0) @RT(0) @RT(7)TaskMid @F @F
@END_Algo

@BEG_Dcl
@RT(16)DclTreeContainer
7
@Var @RT(8)bTimeout @RT(0) @T @F @DT @RT(4)BOOL @RT(0) @T @T @BASIC 0 @F
@F @F
@T
@BEG_Attrib
3 @RT(0) @RT(0) @RT(0)
@END_Attrib
1 0 @F @F @F @F

@Var @RT(13)bOutputActive @RT(0) @T @F @DT @RT(4)BOOL @RT(0) @T @T @BASIC 0 @F
@F @F
@T
@BEG_Attrib
3 @RT(0) @RT(0) @RT(0)
@END_Attrib
1 0 @F @F @F @F

@Var @RT(10)iHeartbeat @RT(0) @T @F @DT @RT(4)DINT @RT(0) @T @T @BASIC 0 @F
@F @F
@T
@BEG_Attrib
3 @RT(0) @RT(0) @RT(0)
@END_Attrib
1 0 @F @F @F @F

@Var @RT(6)bAlive @RT(0) @T @F @DT @RT(4)BOOL @RT(0) @T @T @BASIC 0 @F
@F @F
@T
@BEG_Attrib
3 @RT(0) @RT(0) @RT(0)
@END_Attrib
1 0 @F @F @F @F

@Var @RT(4)iCnt @RT(0) @T @F @DT @RT(4)DINT @RT(0) @T @T @BASIC 0 @F
@F @F
@T
@BEG_Attrib
3 @RT(0) @RT(0) @RT(0)
@END_Attrib
1 0 @F @F @F @F

@Var @RT(5)dummy @RT(0) @T @F @DT @RT(4)DINT @RT(0) @T @T @BASIC 0 @F
@F @F
@T
@BEG_Attrib
3 @RT(0) @RT(0) @RT(0)
@END_Attrib
1 0 @F @F @F @F

@Var @RT(5)sText @RT(0) @T @F @DT @RT(11)STRING(255) @RT(0) @T @T @STRING 0 @F @RT(3)255 @F
@F @F
@T
@BEG_Attrib
3 @RT(0) @RT(0) @RT(0)
@END_Attrib
1 0 @F @F @F @F

@END_Dcl

@END_Export

@BEG_Export

@BEG_Algo
@ALGORITHM @RT(21)aSetHeartbeatInterval @STRUCTURED_TEXT
@RT(0) @RT(0) @RT(0) @F @F
@END_Algo

@BEG_Dcl
@RT(16)DclTreeContainer
1
@Var @RT(9)iInterval @RT(0) @T @F @DT @RT(4)DINT @RT(0) @T @T @BASIC 0 @F
@F @F
@T
@BEG_Attrib
3 @RT(0) @RT(0) @RT(0)
@END_Attrib
1 0 @F @F @F @F

@END_Dcl

@END_Export

@BEG_Export

@BEG_Algo
@POSTUPDATE_ALGORITHM @RT(18)pHeartbeatInterval @STRUCTURED_TEXT
@RT(0) @RT(55)sv_iPanelHeartbeatInterval, sv_iPanelHeartbeatTolerance @RT(9)PU_Task_7 @F @F
@END_Algo

@BEG_Dcl
@RT(16)DclTreeContainer
0
@END_Dcl

@END_Export

@BEG_Export

@BEG_Algo
@POSTUPDATE_ALGORITHM @RT(5)pInit @STRUCTURED_TEXT
@RT(0) @RT(35)sv_bInitDone, sv_bUsePanelHeartbeat @RT(9)PU_Task_3 @F @F
@END_Algo

@BEG_Dcl
@RT(16)DclTreeContainer
0
@END_Dcl

@END_Export

@BEG_Body
@TL(20)
(**************************************** WARNING ********************************************
 *** The KEBA Kemro K2 System including software is not intended for safety control tasks! ***
 ***                       For further information see Comment tab!                        ***
 *********************************************************************************************)

IF sv_iPanelButtonCnt >= cMaxPanelButtons THEN
    IF sv_TraceLevel.bApplication THEN
       sText := CONCAT('ABPanelButtonRegister: number of panel buttons exceeded maximum, omitting button from component %d/%d',
                   DINT_TO_STRING(EventData.Button.iCompId), DINT_TO_STRING(EventData.Button.iIndexId));
       dummy := Print(sText);
    END_IF;
    RETURN;
END_IF;
// This array contains all possible movements/actions that can be used within an HMI application.
// The HMI can read this array in order to dynamically create a HMI machine operation panel on
// the visualisation system.
sv_iPanelButtonCnt := sv_iPanelButtonCnt + 1;
sv_PanelButtons[sv_iPanelButtonCnt] := EventData.Button;

@END_Body

@@@BEG_Comment@@@
@TL(4)
get instance data if start event is received

attention:
taskslot is asigned to make sure that execution is done before evaStart in ABControl.pu
@@@END_Comment@@@

@BEG_Body
@TL(15)
(**************************************** WARNING ********************************************
 *** The KEBA Kemro K2 System including software is not intended for safety control tasks! ***
 ***                       For further information see Comment tab!                        ***
 *********************************************************************************************)

IF (sv_iPanelMovementSelector > 0) THEN
   Button := sv_PanelButtons[sv_iPanelMovementSelector];
   mpbActionVar1 := Button.pbActionVar1;
   mpbActionVar2 := Button.pbActionVar2;
ELSE
   mpbActionVar1 := EMPTY;
   mpbActionVar2 := EMPTY;
END_IF;

@END_Body

@@@BEG_Comment@@@
@TL(0)

@@@END_Comment@@@

@BEG_SfcBody
6 4 5

@BEG_SfcData 2
@StepSeq @RT(4)sseq @F 1
@Loop @RT(4)loop @F 2
@StepSeq @RT(3)seq @F 3
@Loop @RT(4)loop @F 2
@StepSeq @RT(3)seq @F 3
@Step @RT(6)S_Idle @F @T @F @F @RT(0) @F
@AcbCont @RT(7)unnamed @F 2
@Acb @RT(7)Action1 @F @T @RT(1)P @RT(0) @F @F @T @TL(3)
bTimeout := FALSE

@F
@Acb @RT(13)Output_Active @F @T @RT(1)N @RT(0) @F @F @T @TL(6)
IF (mpbActionVar1 = EMPTY OR mpbActionVar2 = EMPTY) THEN
   bOutputActive := FALSE;
ELSE
   bOutputActive := mpbActionVar1^ = TRUE OR mpbActionVar2^ = TRUE;
END_IF;

@F

@Trans @RT(6)Trans1 @F @T @F @F @T @T @TL(3)
bOutputActive = TRUE

@RT(6)Trans1 @F
@Step @RT(14)S_OutputActive @F @F @F @F @RT(0) @F
@AcbCont @RT(7)unnamed @F 2
@Acb @RT(7)Action2 @F @T @RT(1)P @RT(0) @F @F @T @TL(4)
iHeartbeat := sv_iPanelHeartbeat;
bAlive := TRUE;
iCnt := 0;

@F
@Acb @RT(15)Check_Heartbeat @F @T @RT(1)N @RT(0) @F @F @T @TL(24)
IF (mpbActionVar1 = EMPTY AND mpbActionVar2 = EMPTY) THEN
   bOutputActive := FALSE;
ELSE
   bOutputActive := FALSE;
   IF (mpbActionVar1 <> EMPTY) THEN
      bOutputActive := mpbActionVar1^;
   END_IF;
   IF (NOT bOutputActive AND mpbActionVar2 <> EMPTY) THEN
      bOutputActive := mpbActionVar2^;
   END_IF;

   IF (sv_iPanelHeartbeat <> iHeartbeat) THEN
      (* heartbeat counter changed while output active *)
      bAlive := TRUE;
      iHeartbeat := sv_iPanelHeartbeat;
      iCnt := 0;
   ELSE
      iCnt := iCnt + 1;
      IF iCnt > miAliveTicks THEN
         bAlive := FALSE;
      END_IF;
   END_IF;
END_IF;

@F

@Trans @RT(6)Trans3 @F @T @T @T @T @T @TL(2)
NOT bOutputActive

@RT(6)Trans3 @F

@Trans @RT(16)HMI_Disconnected @F @T @F @F @T @T @TL(2)
bAlive = FALSE

@RT(6)Trans2 @F
@Step @RT(9)S_Timeout @F @F @F @F @RT(0) @F
@AcbCont @RT(7)unnamed @F 1
@Acb @RT(8)Reset_IO @F @T @RT(1)N @RT(0) @F @F @T @TL(15)
(* Safety reset *)
IF (mpbActionVar1 <> EMPTY) THEN
   mpbActionVar1^ := FALSE;
END_IF;
IF (mpbActionVar2 <> EMPTY) THEN
   mpbActionVar2^ := FALSE;
END_IF;
IF sv_TraceLevel.bApplication THEN
   sText := CONCAT('HMI timeout, output was reset by heartbeat detection, ticks detected ',
                        DINT_TO_STRING(iCnt),
                        ', maximum ',
                        DINT_TO_STRING(miAliveTicks));
   dummy := Print(sText);
END_IF;

@F

@Trans @RT(6)Trans4 @F @T @T @T @T @T @TL(2)
TRUE

@RT(6)Trans4 @F

@END_SfcData
@SaActions 1
@SaText @RT(7)Action3 1 @TL(2)

@SaTrans 0
@SaExits 0
@END_SfcBody

@@@BEG_Comment@@@
@TL(0)

@@@END_Comment@@@

@BEG_Body
@TL(11)
(* Currently checked in TaskMid *)
iInterval := LINT_TO_DINT(TIME_TO_LINT(GET_TASK_INTERVAL(TaskMid))/1000);

IF sv_iPanelHeartbeatInterval < iInterval THEN
   sv_iPanelHeartbeatInterval := iInterval;
END_IF;

miAliveTicks := (sv_iPanelHeartbeatInterval + sv_iPanelHeartbeatTolerance)/(iInterval);

@END_Body

@@@BEG_Comment@@@
@TL(0)

@@@END_Comment@@@

@BEG_Body
@TL(3)

aSetHeartbeatInterval();

@END_Body

@@@BEG_Comment@@@
@TL(0)

@@@END_Comment@@@

@BEG_Body
@TL(8)

aSetHeartbeatInterval();
IF (sv_bUsePanelHeartbeat) THEN
   START_PROCESS_ALGORITHM(paCheckHeartbeat);
ELSE
   STOP_PROCESS_ALGORITHM(paCheckHeartbeat);
END_IF;

@END_Body

@@@BEG_Comment@@@
@TL(0)

@@@END_Comment@@@
@END_Body

@END_Contents
